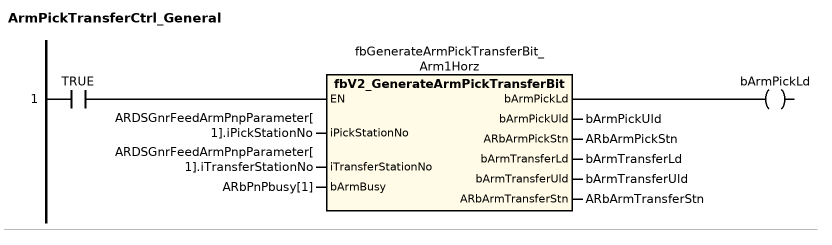
// NETWORK 1
fbGenerateArmPickTransferBit_Arm1Horz(
    iPickStationNo := ARDSGnrFeedArmPnpParameter[1].iPickStationNo,
    iTransferStationNo := ARDSGnrFeedArmPnpParameter[1].iTransferStationNo,
    bArmBusy := ARbPnPbusy[1],
    bArmPickUld => bArmPickUld,
    ARbArmPickStn => ARbArmPickStn,
    bArmTransferLd => bArmTransferLd,
    bArmTransferUld => bArmTransferUld,
    ARbArmTransferStn => ARbArmTransferStn); // fbV2_GenerateArmPickTransferBit
bArmPickLd := fbGenerateArmPickTransferBit_Arm1Horz.bArmPickLd;

END_PROGRAM

// ---- FBs/B_JKS_NewFB_V2/FBP-ArmCtrlFolder/fbV2_GenerateArmPickTransferBit.TcPOU
FUNCTION_BLOCK fbV2_GenerateArmPickTransferBit
VAR_INPUT
	iPickStationNo : INT;
	iTransferStationNo : INT;
	bArmBusy	: BOOL;
END_VAR
VAR_OUTPUT
	bArmPickLd : BOOL;
	bArmPickUld : BOOL;
	ARbArmPickStn : ARRAY [1..iStnQty] OF BOOL;
	bArmTransferLd : BOOL;
	bArmTransferUld : BOOL;
	ARbArmTransferStn : ARRAY [1..iStnQty] OF BOOL;

END_VAR
VAR
	iPickStnFL: INT;
	iClearPickStnFL: INT;
	iTransferStnFL: INT;
	iClearTransferStnFL: INT;
	bArmPickStnFound: BOOL;
	bArmTransferStnFound: BOOL;
END_VAR

(*For Pick Bit Checking*)
IF bArmBusy  THEN

	bArmPickLd := FALSE;
	bArmPickUld := FALSE;
	iClearPickStnFL := 1;
	
		FOR iClearPickStnFL := 1 TO iStnQty DO
			IF iClearPickStnFL >= 1 AND iClearPickStnFL <= iStnQty THEN
					ARbArmPickStn[iClearPickStnFL] := FALSE;
			END_IF
	
		END_FOR
	
	bArmPickStnFound := FALSE;

	IF NOT bArmPickStnFound THEN
		iPickStnFL := 1;
			FOR iPickStnFL := 1 TO iLdStnQty DO
				IF iPickStnFL >= 1 AND iPickStnFL <= iLdStnQty THEN
					 IF iPickStationNo = ARiLdStnID[iLdStnQty] AND ARiLdStnID[iLdStnQty] <> 0 THEN
						bArmPickLd := TRUE;
						bArmPickStnFound := TRUE;
					END_IF
				END_IF
			END_FOR
	END_IF


	IF NOT bArmPickStnFound THEN
		iPickStnFL := 1;
			FOR iPickStnFL := 1 TO iUldStnQty DO
				IF iPickStnFL >= 1 AND iPickStnFL <= iUldStnQty THEN
					 IF iPickStationNo = ARiUldStnID[iUldStnQty] AND ARiUldStnID[iUldStnQty] <> 0 THEN
						bArmPickUld := TRUE;
						bArmPickStnFound := TRUE;
					END_IF
				END_IF
			END_FOR
	END_IF


	IF NOT bArmPickStnFound AND iPickStationNo >= 1 AND iPickStationNo <= iStnQty THEN
		iPickStnFL := 1;
			FOR iPickStnFL := 1 TO iStnQty DO
				IF iPickStnFL >= 1 AND iPickStnFL <= iStnQty THEN
					IF iPickStationNo = iPickStnFL THEN
						ARbArmPickStn[iPickStnFL] := TRUE;
						bArmPickStnFound := TRUE;
					END_IF
				END_IF
			END_FOR
	END_IF

ELSE


	bArmPickLd := FALSE;
	bArmPickUld := FALSE;
	iClearPickStnFL := 1;
	
		FOR iClearPickStnFL := 1 TO iStnQty DO
			IF iClearPickStnFL >= 1 AND iClearPickStnFL <= iStnQty THEN
					ARbArmPickStn[iClearPickStnFL] := FALSE;
			END_IF
	
		END_FOR
	
	bArmPickStnFound := FALSE;


END_IF

(*For Transfer Bit Checking*)

IF bArmBusy  THEN

	bArmTransferLd := FALSE;
	bArmTransferUld := FALSE;
	iClearTransferStnFL := 1;
		FOR iClearTransferStnFL := 1 TO iStnQty DO
			IF iClearTransferStnFL >= 1 AND iClearTransferStnFL <= iStnQty THEN
					ARbArmTransferStn[iClearTransferStnFL] := FALSE;
			END_IF
		END_FOR
	
	bArmTransferStnFound := FALSE;

	IF NOT bArmTransferStnFound THEN
		iTransferStnFL := 1;
			FOR iTransferStnFL := 1 TO iLdStnQty DO
				IF iTransferStnFL >= 1 AND iTransferStnFL <= iLdStnQty THEN
					 IF iTransferStationNo = ARiLdStnID[iLdStnQty] AND ARiLdStnID[iLdStnQty] <> 0 THEN
						bArmTransferLd := TRUE;
						bArmTransferStnFound := TRUE;
					END_IF
				END_IF
			END_FOR
	END_IF


	IF NOT bArmTransferStnFound THEN
		iTransferStnFL := 1;
			FOR iTransferStnFL := 1 TO iUldStnQty DO
				IF iTransferStnFL >= 1 AND iTransferStnFL <= iUldStnQty THEN
					 IF iTransferStationNo = ARiUldStnID[iUldStnQty] AND ARiUldStnID[iUldStnQty] <> 0 THEN
						bArmTransferUld := TRUE;
						bArmTransferStnFound := TRUE;
					END_IF
				END_IF
			END_FOR
	END_IF


	IF NOT bArmTransferStnFound AND iTransferStationNo >= 1 AND iTransferStationNo <= iStnQty THEN
		iTransferStnFL := 1;
			FOR iTransferStnFL := 1 TO iStnQty DO
				IF iTransferStnFL >= 1 AND iTransferStnFL <= iStnQty THEN
					IF iTransferStationNo = iTransferStnFL THEN
						ARbArmTransferStn[iTransferStnFL] := TRUE;
						bArmTransferStnFound := TRUE;
					END_IF
				END_IF
			END_FOR

	END_IF

ELSE


	bArmTransferLd := FALSE;
	bArmTransferUld := FALSE;
	iClearTransferStnFL := 1;
		FOR iClearTransferStnFL := 1 TO iStnQty DO
			IF iClearTransferStnFL >= 1 AND iClearTransferStnFL <= iStnQty THEN
					ARbArmTransferStn[iClearTransferStnFL] := FALSE;
			END_IF
		END_FOR
	
	bArmTransferStnFound := FALSE;

END_IF

END_FUNCTION_BLOCK

// ---- POUs/MainProgram/DataManagement/BasketTotalizer.TcPOU
PROGRAM BasketTotalizer
VAR

END_VAR

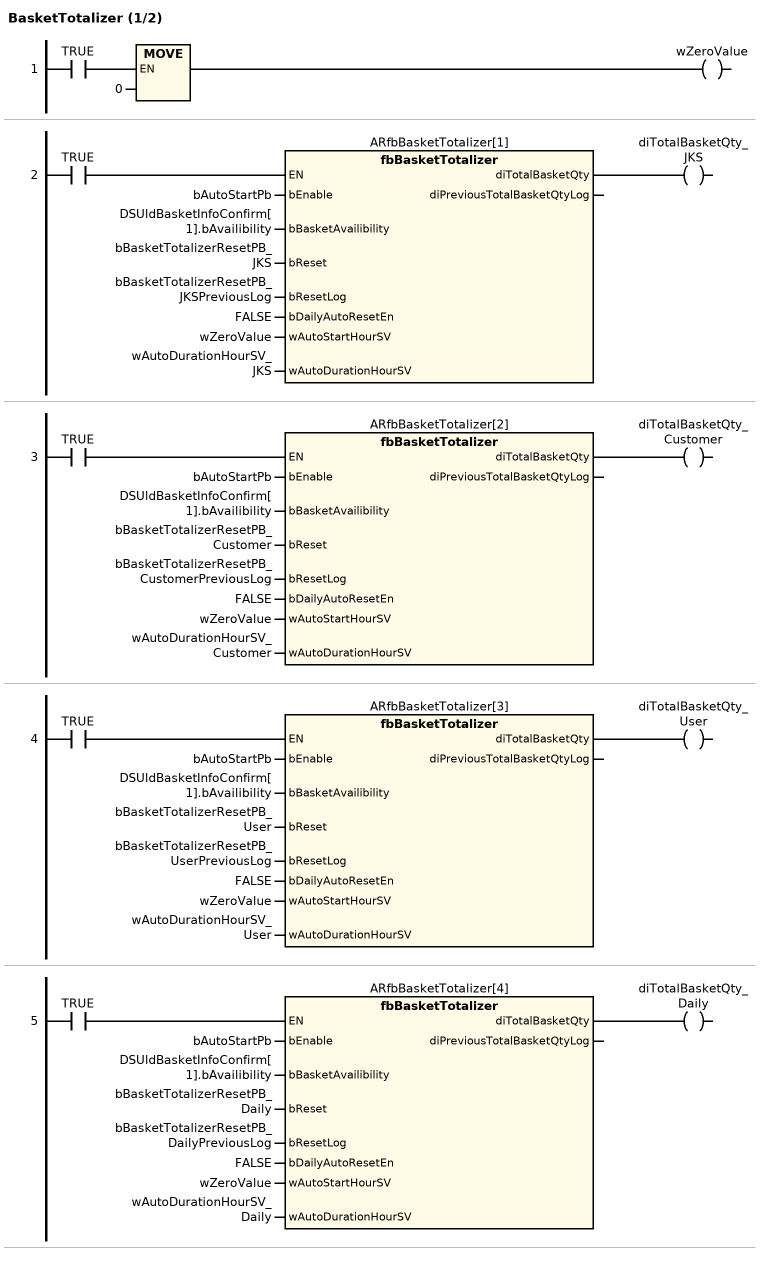
// NETWORK 1
wZeroValue := 0;

// NETWORK 2
ARfbBasketTotalizer[1](
    bEnable := bAutoStartPb,
    bBasketAvailibility := DSUldBasketInfoConfirm[1].bAvailibility,
    bReset := bBasketTotalizerResetPB_JKS,
    bResetLog := bBasketTotalizerResetPB_JKSPreviousLog,
    bDailyAutoResetEn := FALSE,
    wAutoStartHourSV := wZeroValue,
    wAutoDurationHourSV := wAutoDurationHourSV_JKS); // fbBasketTotalizer
diTotalBasketQty_JKS := ARfbBasketTotalizer[1].diTotalBasketQty;

// NETWORK 3
ARfbBasketTotalizer[2](
    bEnable := bAutoStartPb,
    bBasketAvailibility := DSUldBasketInfoConfirm[1].bAvailibility,
    bReset := bBasketTotalizerResetPB_Customer,
    bResetLog := bBasketTotalizerResetPB_CustomerPreviousLog,
    bDailyAutoResetEn := FALSE,
    wAutoStartHourSV := wZeroValue,
    wAutoDurationHourSV := wAutoDurationHourSV_Customer); // fbBasketTotalizer
diTotalBasketQty_Customer := ARfbBasketTotalizer[2].diTotalBasketQty;

// NETWORK 4
ARfbBasketTotalizer[3](
    bEnable := bAutoStartPb,
    bBasketAvailibility := DSUldBasketInfoConfirm[1].bAvailibility,
    bReset := bBasketTotalizerResetPB_User,
    bResetLog := bBasketTotalizerResetPB_UserPreviousLog,
    bDailyAutoResetEn := FALSE,
    wAutoStartHourSV := wZeroValue,
    wAutoDurationHourSV := wAutoDurationHourSV_User); // fbBasketTotalizer
diTotalBasketQty_User := ARfbBasketTotalizer[3].diTotalBasketQty;

// NETWORK 5
ARfbBasketTotalizer[4](
    bEnable := bAutoStartPb,
    bBasketAvailibility := DSUldBasketInfoConfirm[1].bAvailibility,
    bReset := bBasketTotalizerResetPB_Daily,
    bResetLog := bBasketTotalizerResetPB_DailyPreviousLog,
    bDailyAutoResetEn := FALSE,
    wAutoStartHourSV := wZeroValue,
    wAutoDurationHourSV := wAutoDurationHourSV_Daily); // fbBasketTotalizer
diTotalBasketQty_Daily := ARfbBasketTotalizer[4].diTotalBasketQty;

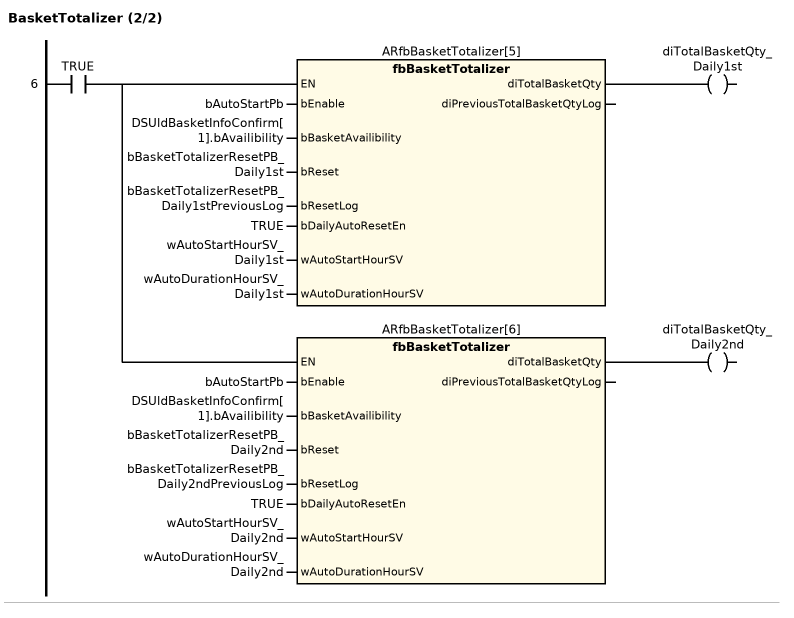
// NETWORK 6
ARfbBasketTotalizer[5](
    bEnable := bAutoStartPb,
    bBasketAvailibility := DSUldBasketInfoConfirm[1].bAvailibility,
    bReset := bBasketTotalizerResetPB_Daily1st,
    bResetLog := bBasketTotalizerResetPB_Daily1stPreviousLog,
    bDailyAutoResetEn := TRUE,
    wAutoStartHourSV := wAutoStartHourSV_Daily1st,
    wAutoDurationHourSV := wAutoDurationHourSV_Daily1st); // fbBasketTotalizer
diTotalBasketQty_Daily1st := ARfbBasketTotalizer[5].diTotalBasketQty;
ARfbBasketTotalizer[6](
    bEnable := bAutoStartPb,
    bBasketAvailibility := DSUldBasketInfoConfirm[1].bAvailibility,
    bReset := bBasketTotalizerResetPB_Daily2nd,
    bResetLog := bBasketTotalizerResetPB_Daily2ndPreviousLog,
    bDailyAutoResetEn := TRUE,
    wAutoStartHourSV := wAutoStartHourSV_Daily2nd,
    wAutoDurationHourSV := wAutoDurationHourSV_Daily2nd); // fbBasketTotalizer
diTotalBasketQty_Daily2nd := ARfbBasketTotalizer[6].diTotalBasketQty;

END_PROGRAM

// ---- FBs/B_JKS_NewFB/FBP-BasketTotalizer/fbBasketTotalizer.TcPOU
FUNCTION_BLOCK fbBasketTotalizer
VAR_INPUT
	bEnable : BOOL; (* Counting will take place if enable*)
	bBasketAvailibility : BOOL;
	bReset : BOOL; 				(*TRUE will reset the total basket qty*)
	bResetLog : BOOL; 			(*TRUE will reset the total basket qty*)
	bDailyAutoResetEn : BOOL; 	(*TRUE if Daily Auto Reset is needed*)
END_VAR

VAR_IN_OUT
	wAutoStartHourSV : WORD; 	(*[Hour: 0..23]*)
	wAutoDurationHourSV : WORD; 	(*[Hour: 0..23]*)

END_VAR

VAR_OUTPUT PERSISTENT
	diTotalBasketQty : DINT;
	diPreviousTotalBasketQtyLog : DINT;
END_VAR
VAR
	TMOUT	: TIME := DEFAULT_ADS_TIMEOUT;(* Max fb execution time *)
	BUSY		: BOOL;
	ERR		: BOOL;
	ERRID		: UDINT;
	TIMESTR	: TIMESTRUCT;(* Local windows system time *)
	NTGetTime: NT_GetTime;
	t1SClockPulse: TON;
	t1SClockPulse_RE: R_TRIG;
	bAutoResetEn_RE: R_TRIG;
	bReset_RE: R_TRIG;
	bResetLog_RE: R_TRIG;
	bCountEn_FE: F_TRIG;
	tResetLog: TON;

	wEndTimeHourSV: WORD;
	bCountEnable: BOOL;
	bEndGTStartFlag: BOOL;
	bEndLTStartFlag: BOOL;

END_VAR

t1SClockPulse(IN:=NOT t1SClockPulse.Q , PT:=t#1s , Q=> , ET=> );
t1SClockPulse_RE(CLK:=t1SClockPulse.Q , Q=> );
NTGetTime(
	NETID:= ,
	START:=t1SClockPulse_RE.Q ,
	TMOUT:=TMOUT ,
	BUSY=>BUSY ,
	ERR=>ERR ,
	ERRID=> ERRID,
	TIMESTR=>TIMESTR );

IF wAutoStartHourSV > 23 THEN
wAutoStartHourSV := 23;
END_IF

IF wAutoDurationHourSV > 23 THEN
wAutoDurationHourSV := 23;
END_IF

IF wAutoDurationHourSV < 1 THEN
wAutoDurationHourSV := 1;
END_IF

IF (wAutoStartHourSV + wAutoDurationHourSV) >= 24 THEN
wEndTimeHourSV :=  (wAutoStartHourSV + wAutoDurationHourSV) - 24;
ELSE
wEndTimeHourSV :=  (wAutoStartHourSV + wAutoDurationHourSV);
END_IF

IF  wAutoStartHourSV < wEndTimeHourSV AND  (wAutoStartHourSV <= TIMESTR.wHour AND wEndTimeHourSV > TIMESTR.wHour) THEN
bEndGTStartFlag := TRUE;
bEndLTStartFlag := FALSE;
bCountEnable := TRUE;
ELSIF wAutoStartHourSV > wEndTimeHourSV AND (wAutoStartHourSV <= TIMESTR.wHour OR wEndTimeHourSV > TIMESTR.wHour) THEN
bEndGTStartFlag := FALSE;
bEndLTStartFlag := TRUE;
bCountEnable := TRUE;
ELSE
bEndGTStartFlag := FALSE;
bEndLTStartFlag := FALSE;
bCountEnable := FALSE;
END_IF


bAutoResetEn_RE(
CLK:=	(((*bEndGTStartFlag AND*) TIMESTR.wHour >= wEndTimeHourSV) OR
		((*bEndLTStartFlag AND*) TIMESTR.wHour >= wEndTimeHourSV AND TIMESTR.wHour < wAutoStartHourSV )) AND bDailyAutoResetEn , Q=> );
bReset_RE(CLK:=bReset , Q=> );
bCountEn_FE(CLK:=bBasketAvailibility , Q=> );
tResetLog(IN:=bResetLog , PT:= t#3s, Q=> , ET=> );
bResetLog_RE(CLK:=tResetLog.Q , Q=> );

IF bReset_RE.Q THEN
diTotalBasketQty := 0;
END_IF

IF bResetLog_RE.Q THEN
diPreviousTotalBasketQtyLog := 0;
END_IF

IF  bAutoResetEn_RE.Q THEN
diPreviousTotalBasketQtyLog := diTotalBasketQty;
diTotalBasketQty := 0;
END_IF
(*
IF  bAutoResetEn_RE.Q OR bReset_RE.Q THEN
diPreviousTotalBasketQtyLog := diTotalBasketQty;
diTotalBasketQty := 0;
END_IF
*)
IF bCountEn_FE.Q AND bEnable AND (NOT bDailyAutoResetEn OR bCountEnable) THEN
diTotalBasketQty := diTotalBasketQty +1;
END_IF

END_FUNCTION_BLOCK

// ---- POUs/MainProgram/DataManagement/MacOperationTimeCtrl.TcPOU
PROGRAM MacOperationTimeCtrl
VAR

END_VAR

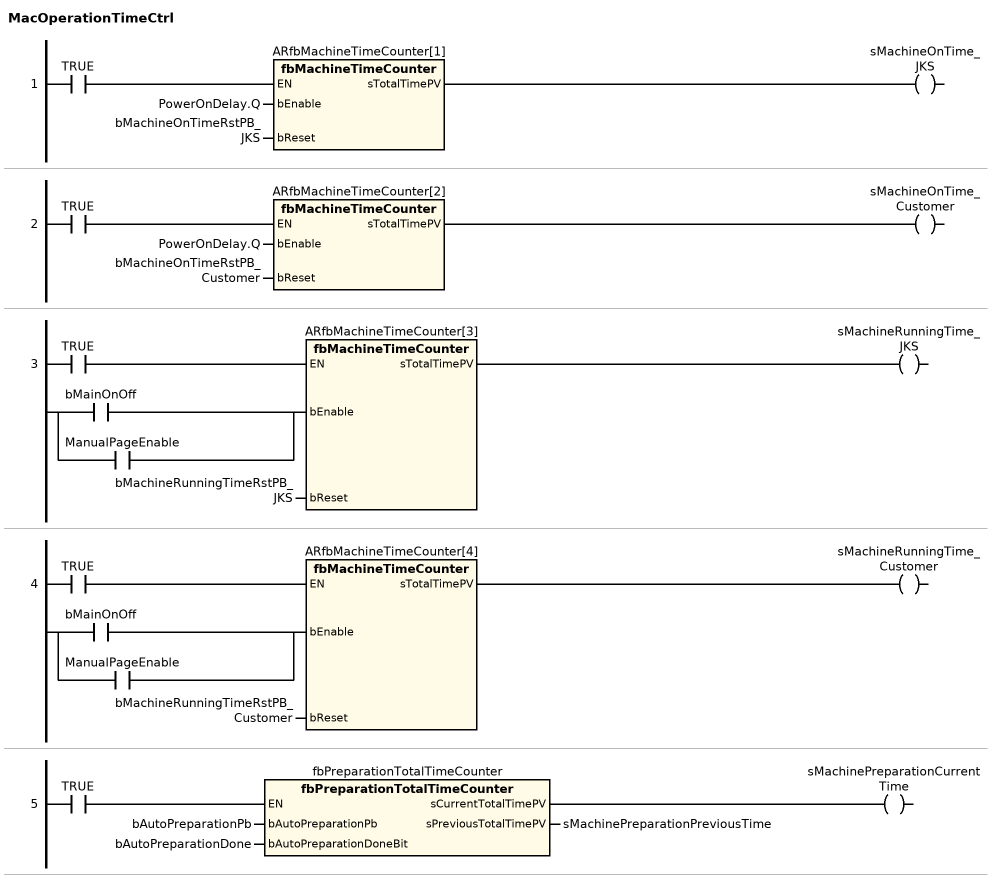
// NETWORK 1
ARfbMachineTimeCounter[1](bEnable := PowerOnDelay.Q, bReset := bMachineOnTimeRstPB_JKS); // fbMachineTimeCounter
sMachineOnTime_JKS := ARfbMachineTimeCounter[1].sTotalTimePV;

// NETWORK 2
ARfbMachineTimeCounter[2](bEnable := PowerOnDelay.Q, bReset := bMachineOnTimeRstPB_Customer); // fbMachineTimeCounter
sMachineOnTime_Customer := ARfbMachineTimeCounter[2].sTotalTimePV;

// NETWORK 3
ARfbMachineTimeCounter[3](bEnable := bMainOnOff OR ManualPageEnable, bReset := bMachineRunningTimeRstPB_JKS); // fbMachineTimeCounter
sMachineRunningTime_JKS := ARfbMachineTimeCounter[3].sTotalTimePV;

// NETWORK 4
ARfbMachineTimeCounter[4](bEnable := bMainOnOff OR ManualPageEnable, bReset := bMachineRunningTimeRstPB_Customer); // fbMachineTimeCounter
sMachineRunningTime_Customer := ARfbMachineTimeCounter[4].sTotalTimePV;

// NETWORK 5
fbPreparationTotalTimeCounter(
    bAutoPreparationPb := bAutoPreparationPb,
    bAutoPreparationDoneBit := bAutoPreparationDone,
    sPreviousTotalTimePV => sMachinePreparationPreviousTime);
sMachinePreparationCurrentTime := fbPreparationTotalTimeCounter.sCurrentTotalTimePV;

END_PROGRAM

// ---- FBs/B_JKS_NewFB/FBP-MachineOperationTimeCounter/fbMachineTimeCounter.TcPOU
FUNCTION_BLOCK fbMachineTimeCounter
VAR_INPUT
	bEnable		: BOOL;
	bReset		: BOOL;
END_VAR

VAR_OUTPUT
	sTotalTimePV	: STRING;
END_VAR
VAR

	TON1			: TON;
	TON2			: TON;
	FBTRIG			: R_TRIG;
	FB1TRIG		: R_TRIG;
	step				: INT;

	Second				: DINT;

END_VAR
VAR PERSISTENT
	Counter				: DINT;
	Minute				: DINT;
	Hour				: DINT;
	Day					: DINT;
END_VAR

TON1(IN:=(bEnable AND NOT TON2.Q) , PT:=T#0.5S , Q=> , ET=> );
TON2(IN:=TON1.Q , PT:=T#0.5S , Q=> , ET=> );
FB1TRIG(CLK:=bReset , Q=> );

IF bEnable THEN
	FBTRIG(CLK:=TON2.Q , Q=> );
END_IF

IF FB1TRIG.Q THEN
	Counter		:= 0;
	Second		:= 0;
	Minute		:= 0;
	Hour		:= 0;
	Day			:= 0;
END_IF

IF bEnable AND FBTRIG.Q THEN
	Second := Second + 1;
END_IF

IF bEnable AND Second >= 60 THEN
	Minute := MInute + 1;
	Second := 0;
END_IF

IF bEnable AND Minute >= 60 THEN
	Hour := hour + 1;
	Minute := 0;
END_IF

IF bEnable AND Hour >= 24 THEN
	Day := Day +1;
	Hour := 0;
END_IF

sTotalTimePV := CONCAT(DINT_TO_STRING(Day),':');

IF Hour < 10 THEN
sTotalTimePV :=CONCAT(sTotalTimePV,'0');
sTotalTimePV :=CONCAT(sTotalTimePV,DINT_TO_STRING(Hour));
ELSE
sTotalTimePV :=CONCAT(sTotalTimePV,DINT_TO_STRING(Hour));
END_IF

sTotalTimePV := CONCAT(sTotalTimePV,':');

IF Minute < 10 THEN
sTotalTimePV :=CONCAT(sTotalTimePV,'0');
sTotalTimePV :=CONCAT(sTotalTimePV,DINT_TO_STRING(Minute));
ELSE
sTotalTimePV :=CONCAT(sTotalTimePV,DINT_TO_STRING(Minute));
END_IF

sTotalTimePV := CONCAT(sTotalTimePV,':');

IF Second < 10 THEN
sTotalTimePV := CONCAT(sTotalTimePV,'0');
sTotalTimePV := CONCAT(sTotalTimePV,DINT_TO_STRING(Second));
ELSE
sTotalTimePV := CONCAT(sTotalTimePV,DINT_TO_STRING(Second));
END_IF

END_FUNCTION_BLOCK

// ---- POUs/MainProgram/DataManagement/RTClockCtrl.TcPOU
PROGRAM RTClockCtrl
VAR

(*Local*)
	TMOUT				: TIME := DEFAULT_ADS_TIMEOUT;(* Max fb execution time *)
	BUSY				: BOOL;
	ERR				: BOOL;
	ERRID				: UDINT;
	TIMESTR			: TIMESTRUCT;(* Local windows system time *)
	NTGetTime			: NT_GetTime;
	t1SClockPulse		: TON;
	t1SClockPulse_RE	: R_TRIG;

(*Global*)

END_VAR

t1SClockPulse(IN:=NOT t1SClockPulse.Q , PT:=t#1s , Q=> , ET=> );
t1SClockPulse_RE(CLK:=t1SClockPulse.Q , Q=> );
NTGetTime(
	NETID:= , 
	START:=t1SClockPulse_RE.Q ,
	TMOUT:=TMOUT ,
	BUSY=>BUSY ,
	ERR=>ERR ,
	ERRID=> ERRID,
	TIMESTR=>TIMESTR );


IF TIMESTR.wYear >= wShutDownYear AND TIMESTR.wMonth >= wShutDownMonth AND TIMESTR.wDay >= wShutDownDay AND NOT bMcShutDownDisable THEN
bSystemError := TRUE;
END_IF

IF bMcShutDownDisable THEN
bSystemError := FALSE;
END_IF

END_PROGRAM

// ---- POUs/MainProgram/DataManagement/StnBasketTotalizer.TcPOU
PROGRAM StnBasketTotalizer
VAR

END_VAR

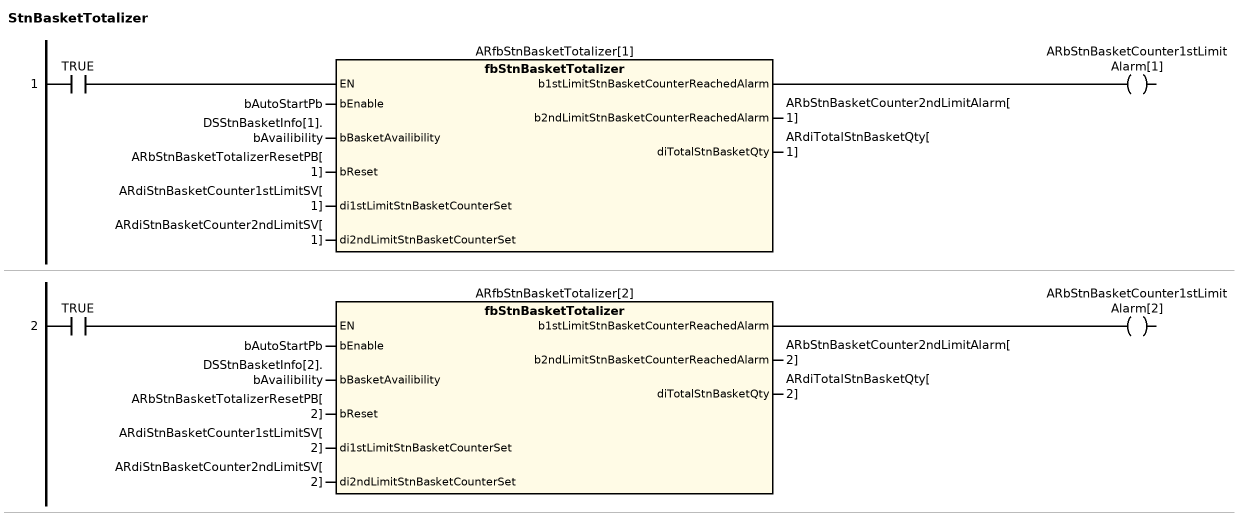
// NETWORK 1
ARfbStnBasketTotalizer[1](
    bEnable := bAutoStartPb,
    bBasketAvailibility := DSStnBasketInfo[1].bAvailibility,
    bReset := ARbStnBasketTotalizerResetPB[1],
    di1stLimitStnBasketCounterSet := ARdiStnBasketCounter1stLimitSV[1],
    di2ndLimitStnBasketCounterSet := ARdiStnBasketCounter2ndLimitSV[1],
    b2ndLimitStnBasketCounterReachedAlarm => ARbStnBasketCounter2ndLimitAlarm[1],
    diTotalStnBasketQty => ARdiTotalStnBasketQty[1]); // fbStnBasketTotalizer
ARbStnBasketCounter1stLimitAlarm[1] := ARfbStnBasketTotalizer[1].b1stLimitStnBasketCounterReachedAlarm;

// NETWORK 2
ARfbStnBasketTotalizer[2](
    bEnable := bAutoStartPb,
    bBasketAvailibility := DSStnBasketInfo[2].bAvailibility,
    bReset := ARbStnBasketTotalizerResetPB[2],
    di1stLimitStnBasketCounterSet := ARdiStnBasketCounter1stLimitSV[2],
    di2ndLimitStnBasketCounterSet := ARdiStnBasketCounter2ndLimitSV[2],
    b2ndLimitStnBasketCounterReachedAlarm => ARbStnBasketCounter2ndLimitAlarm[2],
    diTotalStnBasketQty => ARdiTotalStnBasketQty[2]); // fbStnBasketTotalizer
ARbStnBasketCounter1stLimitAlarm[2] := ARfbStnBasketTotalizer[2].b1stLimitStnBasketCounterReachedAlarm;

END_PROGRAM

// ---- FBs/B_JKS_NewFB/FBP-BasketTotalizer/fbStnBasketTotalizer.TcPOU
FUNCTION_BLOCK fbStnBasketTotalizer
VAR_INPUT
	bEnable : BOOL; (* Counting will take place if enable*)
	bBasketAvailibility : BOOL;
	bReset : BOOL; 				(*TRUE will reset the total Stn basket Qty*)

END_VAR

VAR_OUTPUT
	b1stLimitStnBasketCounterReachedAlarm: BOOL;
	b2ndLimitStnBasketCounterReachedAlarm: BOOL;

END_VAR

VAR_IN_OUT
	di1stLimitStnBasketCounterSet : DINT;
	di2ndLimitStnBasketCounterSet : DINT;
END_VAR

VAR_OUTPUT PERSISTENT
	diTotalStnBasketQty : DINT;
END_VAR

VAR
	bReset_RE: R_TRIG;
	bCountEn_FE: F_TRIG;

END_VAR

IF di1stLimitStnBasketCounterSet > 9999 THEN
di1stLimitStnBasketCounterSet := 9999;
END_IF

IF di1stLimitStnBasketCounterSet < 1 THEN
di1stLimitStnBasketCounterSet := 1;
END_IF

IF di2ndLimitStnBasketCounterSet > 9999 THEN
di2ndLimitStnBasketCounterSet := 9999;
END_IF

IF di2ndLimitStnBasketCounterSet < 2 THEN
di2ndLimitStnBasketCounterSet := 2;
END_IF

IF di2ndLimitStnBasketCounterSet = di1stLimitStnBasketCounterSet THEN
di1stLimitStnBasketCounterSet := di2ndLimitStnBasketCounterSet - 1 ;
END_IF

IF di2ndLimitStnBasketCounterSet <= di1stLimitStnBasketCounterSet THEN
di2ndLimitStnBasketCounterSet := di1stLimitStnBasketCounterSet + 1 ;
END_IF


bReset_RE(CLK:=bReset , Q=> );
bCountEn_FE(CLK:=bBasketAvailibility , Q=> );

IF bReset_RE.Q THEN
diTotalStnBasketQty := 0;
END_IF

IF bCountEn_FE.Q AND bEnable THEN
diTotalStnBasketQty := diTotalStnBasketQty +1;
END_IF

IF bEnable AND diTotalStnBasketQty >= di1stLimitStnBasketCounterSet THEN
	b1stLimitStnBasketCounterReachedAlarm := TRUE;
ELSE
	b1stLimitStnBasketCounterReachedAlarm := FALSE;
END_IF

IF bEnable AND diTotalStnBasketQty >= di2ndLimitStnBasketCounterSet THEN
	b2ndLimitStnBasketCounterReachedAlarm := TRUE;
ELSE
	b2ndLimitStnBasketCounterReachedAlarm := FALSE;
END_IF

END_FUNCTION_BLOCK

// ---- POUs/MainProgram/Csv/Batch_Number_counter.TcPOU
PROGRAM Batch_Number_counter
VAR
	R_TRIG1	: R_TRIG;
END_VAR

(*Time Log to create an unique file number for the Report file name*)

(*Time_log := F_jx_TS_TO_TIME_STRING;*)

R_TRIG1(CLK:=AR2sDSCv_LdConfirmBasketInfo[1,4].bAvailibility  , Q=> );

(*DSArmBasketInfo[1].bAvailibility*)
IF R_TRIG1.Q  THEN
	iProgBatchTotal:=iProgBatchTotal+1;
	AR2sDSCv_LdConfirmBasketInfo[1,4].sReservedInt:=INT_TO_STRING(iProgBatchTotal);

END_IF
IF iProgBatchTotal > 30000 THEN
iProgBatchTotal:=0;
END_IF

END_PROGRAM

// ---- POUs/MainProgram/Csv/Csv_Report_Ctrl.TcPOU
PROGRAM Csv_Report_Ctrl
VAR
	bEn	:	BOOL;
	bReset : BOOL;
	
	bIdleFlag : BOOL;
	bProgressFlag : BOOL;
	
	bErrorFlag : BOOL;
	iErrorCaseId : INT;
	bClearErrorLog : BOOL;
	
	bError			: BOOL;
	

	tReportCsvEn_Ld: TON;
	bReportCsvWriteRE_Ld: R_TRIG;
	bErrorCsvLd			: BOOL;
	
	tReportCsvEn_Stn: ARRAY [1..iStnQty] OF TON;	
	bReportCsvWriteRE_Stn: ARRAY [1..iStnQty] OF R_TRIG;
	bErrorCsvStn		: ARRAY [1..13] OF BOOL;
	
	tReportCsvEn_Uld: TON;
	bReportCsvWriteRE_Uld: R_TRIG;
	bErrorCsvUld			: BOOL;
	
	CKKTEST: ARRAY [1..13] OF BOOL;
	sReportName : STRING;
	
	bUsFreqChange: ARRAY [1..iStnQty] OF R_TRIG;
	
	tLd			: TON;
	tStn1		: TON;
	tStn2		: TON;
	tStn3		: TON;
	tStn4		: TON;
	tStn5		: TON;
	tStn6		: TON;
	tStn7		: TON;
	tStn8		: TON;
	tStn9		: TON;
	tStn10		: TON;
	tStn11		: TON;
	tStn12		: TON;
	tStn13		: TON;
	bCsvShutdownRequestFlag: BOOL;
	bCsvReadyToShutdownFlag: BOOL;
	R_TRIG1: R_TRIG;
	test13: BOOL;
	start: BOOL;
	sPath: STRING(255);
	sPath1: STRING(255);
	
		fbFileRename    : FB_FileRename;
		sNetId          : T_AmsNetId;
        sOldName        : T_MaxString;
        sNewName        : T_MaxString;
        ePath           : E_OpenPath := PATH_GENERIC;          (* Default: generic file path*)
        bExecute        : BOOL;
        tTimeout        : TIME;
	bRename: BOOL;
	bReportCsvWriteLdHolding: BOOL;
	tReportCsvWriteLdHolding: TON;
	ARbReportCsvWriteStnHolding : ARRAY [1..iStnQty] OF BOOL;
	ARtReportCsvWriteStnHolding : ARRAY [1..iStnQty] OF TON;
	bReportCsvWriteUldHolding: BOOL;
	tReportCsvWriteUldHolding: TON;
END_VAR

//tReportCsvEn_Ld	    (IN:=dsMcCarrierInfo.ARLd[1].bAvailability , PT:=T#2S ,Q=> , ET=> );
//tReportCsvEn_Stn[1]	(IN:=dsMcCarrierInfo.ARStn[1].iEstTotalProcessTimeEV > 0 AND dsMcCarrierInfo.ARStn[1].iEstTotalProcessTimeEV < 15 , PT:=T#1S ,Q=> , ET=> );
//tReportCsvEn_Stn[2]	(IN:=dsMcCarrierInfo.ARStn[2].iEstTotalProcessTimeEV > 0 AND dsMcCarrierInfo.ARStn[2].iEstTotalProcessTimeEV < 15 , PT:=T#1S ,Q=> , ET=> );
//tReportCsvEn_Stn[3]	(IN:=dsMcCarrierInfo.ARStn[3].iEstTotalProcessTimeEV > 0 AND dsMcCarrierInfo.ARStn[3].iEstTotalProcessTimeEV < 15 , PT:=T#1S ,Q=> , ET=> );
//tReportCsvEn_Stn[4]	(IN:=dsMcCarrierInfo.ARStn[4].iEstTotalProcessTimeEV > 0 AND dsMcCarrierInfo.ARStn[4].iEstTotalProcessTimeEV < 15 , PT:=T#1S ,Q=> , ET=> );
//tReportCsvEn_Stn[5]	(IN:=dsMcCarrierInfo.ARStn[5].iEstTotalProcessTimeEV > 0 AND dsMcCarrierInfo.ARStn[5].iEstTotalProcessTimeEV < 15 , PT:=T#1S ,Q=> , ET=> );
//tReportCsvEn_Uld	(IN:=dsMcCarrierInfo.ARUld[1].bAvailability , PT:=T#1S ,Q=> , ET=> );

tLD(IN:=AR2sDSCv_LdConfirmBasketInfo[1,4].bAvailibility , PT:=T#1S , Q=> , ET=> );
tStn1(IN:=ARDsStnSeqProcessCtrl[1].Out_iTotalProcessTimeEV >0 AND ARDsStnSeqProcessCtrl[1].Out_iTotalProcessTimeEV <10 , PT:=T#1S , Q=> , ET=> );
tStn2(IN:=ARDsStnSeqProcessCtrl[2].Out_iTotalProcessTimeEV >0 AND ARDsStnSeqProcessCtrl[2].Out_iTotalProcessTimeEV <10 , PT:=T#1s , Q=> , ET=> );
tStn3(IN:=ARDsStnSeqProcessCtrl[3].Out_iTotalProcessTimeEV >0 AND ARDsStnSeqProcessCtrl[3].Out_iTotalProcessTimeEV <10 , PT:=T#1s , Q=> , ET=> );
tStn4(IN:=ARDsStnSeqProcessCtrl[4].Out_iTotalProcessTimeEV >0 AND ARDsStnSeqProcessCtrl[4].Out_iTotalProcessTimeEV <10  , PT:=T#1s , Q=> , ET=> );
tStn5(IN:=ARDsStnSeqProcessCtrl[5].Out_iTotalProcessTimeEV >0 AND ARDsStnSeqProcessCtrl[5].Out_iTotalProcessTimeEV <10 , PT:=T#1s , Q=> , ET=> );
tStn6(IN:=ARDsStnSeqProcessCtrl[6].Out_iTotalProcessTimeEV >0 AND ARDsStnSeqProcessCtrl[6].Out_iTotalProcessTimeEV <10 , PT:=T#1s , Q=> , ET=> );
tStn7(IN:=ARDsStnSeqProcessCtrl[7].Out_iTotalProcessTimeEV >0 AND ARDsStnSeqProcessCtrl[7].Out_iTotalProcessTimeEV <10 , PT:=T#1s , Q=> , ET=> );
tStn8(IN:=ARDsStnSeqProcessCtrl[8].Out_iTotalProcessTimeEV >0 AND ARDsStnSeqProcessCtrl[8].Out_iTotalProcessTimeEV <10 , PT:=T#1s , Q=> , ET=> );
tStn9(IN:=ARDsStnSeqProcessCtrl[9].Out_iTotalProcessTimeEV >0 AND ARDsStnSeqProcessCtrl[9].Out_iTotalProcessTimeEV <10 , PT:=T#1s, Q=> , ET=> );
tStn10(IN:=ARDsStnSeqProcessCtrl[10].Out_iTotalProcessTimeEV >0 AND ARDsStnSeqProcessCtrl[10].Out_iTotalProcessTimeEV <10 , PT:=T#1s , Q=> , ET=> );
tStn11(IN:=ARDsStnSeqProcessCtrl[11].Out_iTotalProcessTimeEV >0 AND ARDsStnSeqProcessCtrl[11].Out_iTotalProcessTimeEV <10 , PT:=T#1s , Q=> , ET=> );
tStn12(IN:=ARDsStnSeqProcessCtrl[12].Out_iTotalProcessTimeEV >0 AND ARDsStnSeqProcessCtrl[12].Out_iTotalProcessTimeEV <10 , PT:=T#1s , Q=> , ET=> );
tStn13(IN:=AR2sDSCv_UldConfirmBasketInfo[1,1].bAvailibility  , PT:=T#1S , Q=> , ET=> );


bUsFreqChange[1](CLK:=ARbDO[eY10001_Stn01UltrasonicGeneratorFrequencyChange]  , Q=> );
bUsFreqChange[2](CLK:=ARbDO[eY10002_Stn02UltrasonicGeneratorFrequencyChange]  , Q=> );
bUsFreqChange[4](CLK:=ARbDO[eY10003_Stn04UltrasonicGeneratorFrequencyChange]  , Q=> );
bUsFreqChange[5](CLK:=ARbDO[eY10004_Stn05UltrasonicGeneratorFrequencyChange]  , Q=> );
bUsFreqChange[7](CLK:=ARbDO[eY10005_Stn07UltrasonicGeneratorFrequencyChange]  , Q=> );
bUsFreqChange[8](CLK:=ARbDO[eY10006_Stn08UltrasonicGeneratorFrequencyChange]  , Q=> );



sLdtittle := CONCAT('_',DSLocalSystemTimeML.sCurrentDate_General);
sLdtittle := CONCAT(AR2sDSCv_LdConfirmBasketInfo[1,4].ARsBarcodeData[1],sLdtittle);
sLdtittle := CONCAT('-',sLdtittle);
sLdtittle := CONCAT(AR2sDSCv_LdConfirmBasketInfo[1,4].ARsBarcodeData[2],sLdtittle);
sLdtittle := CONCAT('-',sLdtittle);
sLdtittle := CONCAT(AR2sDSCv_LdConfirmBasketInfo[1,4].ARsBarcodeData[3],sLdtittle);
sLdtittle := CONCAT('-',sLdtittle);
sLdtittle := CONCAT(AR2sDSCv_LdConfirmBasketInfo[1,4].sReservedInt,sLdtittle);

tReportCsvWriteLdHolding(IN:=bReportCsvWriteLdHolding , PT:=T#3S , Q=> , ET=> );
IF bReportCsvWriteRE_Ld.Q THEN bReportCsvWriteLdHolding := TRUE; END_IF
IF tReportCsvWriteLdHolding.Q THEN	bReportCsvWriteLdHolding := FALSE; END_IF

// Loading pick
bReportCsvWriteRE_Ld (CLK:=tLD.Q OR CKKTEST[1] , Q=> );

IF bReportCsvWriteRE_Ld.Q  THEN
	FNbCsvWriteToBuffer(
						iStationId				:=	79 , 
						sFilename				:=	sLdtittle , 
						eCsvActionType			:=	eCsvNewFile_CarrierReport , 
						udiCsvMRBCount			=> 	udiCsvMRBCount, 
						udiCsvMRBUsagePercent	=>	udiCsvMRBUsagePercent , 
						bError					=>	bErrorCsvLd );
END_IF


sStn1tittle := CONCAT('_',DSLocalSystemTimeML.sCurrentDate_General);
sStn1tittle := CONCAT(DSStnBasketInfo[1].ARsBarcodeData[1],sStn1tittle);
sStn1tittle := CONCAT('-',sStn1tittle);
sStn1tittle := CONCAT(DSStnBasketInfo[1].ARsBarcodeData[2],sStn1tittle);
sStn1tittle := CONCAT('-',sStn1tittle);
sStn1tittle := CONCAT(DSStnBasketInfo[1].ARsBarcodeData[3],sStn1tittle);
sStn1tittle := CONCAT('-',sStn1tittle);
sStn1tittle := CONCAT(DSStnBasketInfo[1].sReservedInt,sStn1tittle);

ARtReportCsvWriteStnHolding[1](IN:=ARbReportCsvWriteStnHolding[1] , PT:=T#3S , Q=> , ET=> );
IF bReportCsvWriteRE_Stn[1].Q 		THEN 	ARbReportCsvWriteStnHolding[1] := TRUE; END_IF
IF ARtReportCsvWriteStnHolding[1].Q THEN	ARbReportCsvWriteStnHolding[1] := FALSE; END_IF

// Station 1
bReportCsvWriteRE_Stn[1] (CLK:=tStn1.Q OR GeneratorComparison.ARUpdate_bIntAddress[1] OR CKKTEST[2]    , Q=> );

IF  bReportCsvWriteRE_Stn[1].Q THEN
	FNbCsvWriteToBuffer(
						iStationId				:=	1 , 
						sFilename				:=	sStn1tittle, 
						eCsvActionType			:=	eCsvLogData_CarrierReport , 
						udiCsvMRBCount			=> 	udiCsvMRBCount, 
						udiCsvMRBUsagePercent	=>	udiCsvMRBUsagePercent , 
						bError					=>	bErrorCsvStn[1] );
END_IF


sStn2tittle := CONCAT('_',DSLocalSystemTimeML.sCurrentDate_General);
sStn2tittle := CONCAT(DSStnBasketInfo[2].ARsBarcodeData[1],sStn2tittle);
sStn2tittle := CONCAT('-',sStn2tittle);
sStn2tittle := CONCAT(DSStnBasketInfo[2].ARsBarcodeData[2],sStn2tittle);
sStn2tittle := CONCAT('-',sStn2tittle);
sStn2tittle := CONCAT(DSStnBasketInfo[2].ARsBarcodeData[3],sStn2tittle);
sStn2tittle := CONCAT('-',sStn2tittle);
sStn2tittle := CONCAT(DSStnBasketInfo[2].sReservedInt,sStn2tittle);

ARtReportCsvWriteStnHolding[2](IN:=ARbReportCsvWriteStnHolding[2] , PT:=T#3S , Q=> , ET=> );
IF bReportCsvWriteRE_Stn[2].Q 		THEN 	ARbReportCsvWriteStnHolding[2] := TRUE; END_IF
IF ARtReportCsvWriteStnHolding[2].Q THEN	ARbReportCsvWriteStnHolding[2] := FALSE; END_IF

// Station 2
bReportCsvWriteRE_Stn[2] (CLK:=tStn2.Q OR GeneratorComparison.ARUpdate_bIntAddress[2] OR CKKTEST[3]  , Q=> );

IF  bReportCsvWriteRE_Stn[2].Q THEN
	FNbCsvWriteToBuffer(
						iStationId				:=	2 , 
						sFilename				:=	sStn2tittle , 
						eCsvActionType			:=	eCsvLogData_CarrierReport , 
						udiCsvMRBCount			=> 	udiCsvMRBCount, 
						udiCsvMRBUsagePercent	=>	udiCsvMRBUsagePercent , 
						bError					=>	bErrorCsvStn[2] );
END_IF


sStn3tittle := CONCAT('_',DSLocalSystemTimeML.sCurrentDate_General);
sStn3tittle := CONCAT(DSStnBasketInfo[3].ARsBarcodeData[1],sStn3tittle);
sStn3tittle := CONCAT('-',sStn3tittle);
sStn3tittle := CONCAT(DSStnBasketInfo[3].ARsBarcodeData[2],sStn3tittle);
sStn3tittle := CONCAT('-',sStn3tittle);
sStn3tittle := CONCAT(DSStnBasketInfo[3].ARsBarcodeData[3],sStn3tittle);
sStn3tittle := CONCAT('-',sStn3tittle);
sStn3tittle := CONCAT(DSStnBasketInfo[3].sReservedInt,sStn3tittle);

ARtReportCsvWriteStnHolding[3](IN:=ARbReportCsvWriteStnHolding[3] , PT:=T#3S , Q=> , ET=> );
IF bReportCsvWriteRE_Stn[3].Q 		THEN 	ARbReportCsvWriteStnHolding[3] := TRUE; END_IF
IF ARtReportCsvWriteStnHolding[3].Q THEN	ARbReportCsvWriteStnHolding[3] := FALSE; END_IF

// Station 3
bReportCsvWriteRE_Stn[3] (CLK:=tStn3.Q OR GeneratorComparison.ARUpdate_bIntAddress[3] OR CKKTEST[4]  , Q=> );

IF  bReportCsvWriteRE_Stn[3].Q THEN
	FNbCsvWriteToBuffer(
						iStationId				:=	3 , 
						sFilename				:=	sStn3tittle , 
						eCsvActionType			:=	eCsvLogData_CarrierReport , 
						udiCsvMRBCount			=> 	udiCsvMRBCount, 
						udiCsvMRBUsagePercent	=>	udiCsvMRBUsagePercent , 
						bError					=>	bErrorCsvStn[3] );
END_IF


sStn4tittle := CONCAT('_',DSLocalSystemTimeML.sCurrentDate_General);
sStn4tittle := CONCAT(DSStnBasketInfo[4].ARsBarcodeData[1],sStn4tittle);
sStn4tittle := CONCAT('-',sStn4tittle);
sStn4tittle := CONCAT(DSStnBasketInfo[4].ARsBarcodeData[2],sStn4tittle);
sStn4tittle := CONCAT('-',sStn4tittle);
sStn4tittle := CONCAT(DSStnBasketInfo[4].ARsBarcodeData[3],sStn4tittle);
sStn4tittle := CONCAT('-',sStn4tittle);
sStn4tittle := CONCAT(DSStnBasketInfo[4].sReservedInt,sStn4tittle);

ARtReportCsvWriteStnHolding[4](IN:=ARbReportCsvWriteStnHolding[4] , PT:=T#3S , Q=> , ET=> );
IF bReportCsvWriteRE_Stn[4].Q 		THEN 	ARbReportCsvWriteStnHolding[4] := TRUE; END_IF
IF ARtReportCsvWriteStnHolding[4].Q THEN	ARbReportCsvWriteStnHolding[4] := FALSE; END_IF

// Station 4
bReportCsvWriteRE_Stn[4] (CLK:=tStn4.Q OR GeneratorComparison.ARUpdate_bIntAddress[4] OR CKKTEST[5]  , Q=> );

IF  bReportCsvWriteRE_Stn[4].Q THEN
	FNbCsvWriteToBuffer(
						iStationId				:=	4 , 
						sFilename				:=	sStn4tittle , 
						eCsvActionType			:=	eCsvLogData_CarrierReport , 
						udiCsvMRBCount			=> 	udiCsvMRBCount, 
						udiCsvMRBUsagePercent	=>	udiCsvMRBUsagePercent , 
						bError					=>	bErrorCsvStn[4] );
END_IF


sStn5tittle := CONCAT('_',DSLocalSystemTimeML.sCurrentDate_General);
sStn5tittle := CONCAT(DSStnBasketInfo[5].ARsBarcodeData[1],sStn5tittle);
sStn5tittle := CONCAT('-',sStn5tittle);
sStn5tittle := CONCAT(DSStnBasketInfo[5].ARsBarcodeData[2],sStn5tittle);
sStn5tittle := CONCAT('-',sStn5tittle);
sStn5tittle := CONCAT(DSStnBasketInfo[5].ARsBarcodeData[3],sStn5tittle);
sStn5tittle := CONCAT('-',sStn5tittle);
sStn5tittle := CONCAT(DSStnBasketInfo[5].sReservedInt,sStn5tittle);

ARtReportCsvWriteStnHolding[5](IN:=ARbReportCsvWriteStnHolding[5] , PT:=T#3S , Q=> , ET=> );
IF bReportCsvWriteRE_Stn[5].Q 		THEN 	ARbReportCsvWriteStnHolding[5] := TRUE; END_IF
IF ARtReportCsvWriteStnHolding[5].Q THEN	ARbReportCsvWriteStnHolding[5] := FALSE; END_IF

// Station 5
bReportCsvWriteRE_Stn[5] (CLK:=tStn5.Q OR GeneratorComparison.ARUpdate_bIntAddress[5] OR CKKTEST[6]  , Q=> );

IF  bReportCsvWriteRE_Stn[5].Q THEN
	FNbCsvWriteToBuffer(
						iStationId				:=	5 , 
						sFilename				:=	sStn5tittle, 
						eCsvActionType			:=	eCsvLogData_CarrierReport , 
						udiCsvMRBCount			=> 	udiCsvMRBCount, 
						udiCsvMRBUsagePercent	=>	udiCsvMRBUsagePercent , 
						bError					=>	bErrorCsvStn[5] );
END_IF


sStn6tittle := CONCAT('_',DSLocalSystemTimeML.sCurrentDate_General);
sStn6tittle := CONCAT(DSStnBasketInfo[6].ARsBarcodeData[1],sStn6tittle);
sStn6tittle := CONCAT('-',sStn6tittle);
sStn6tittle := CONCAT(DSStnBasketInfo[6].ARsBarcodeData[2],sStn6tittle);
sStn6tittle := CONCAT('-',sStn6tittle);
sStn6tittle := CONCAT(DSStnBasketInfo[6].ARsBarcodeData[3],sStn6tittle);
sStn6tittle := CONCAT('-',sStn6tittle);
sStn6tittle := CONCAT(DSStnBasketInfo[6].sReservedInt,sStn6tittle);

ARtReportCsvWriteStnHolding[6](IN:=ARbReportCsvWriteStnHolding[6] , PT:=T#3S , Q=> , ET=> );
IF bReportCsvWriteRE_Stn[6].Q 		THEN 	ARbReportCsvWriteStnHolding[6] := TRUE; END_IF
IF ARtReportCsvWriteStnHolding[6].Q THEN	ARbReportCsvWriteStnHolding[6] := FALSE; END_IF

// Station 6
bReportCsvWriteRE_Stn[6] (CLK:=tStn6.Q OR GeneratorComparison.ARUpdate_bIntAddress[6] OR CKKTEST[7]  , Q=> );

IF bReportCsvWriteRE_Stn[6].Q THEN
	FNbCsvWriteToBuffer(
						iStationId				:=	6 , 
						sFilename				:=	sStn6tittle, 
						eCsvActionType			:=	eCsvLogData_CarrierReport , 
						udiCsvMRBCount			=> 	udiCsvMRBCount, 
						udiCsvMRBUsagePercent	=>	udiCsvMRBUsagePercent , 
						bError					=>	bErrorCsvStn[6] );
END_IF


sStn7tittle := CONCAT('_',DSLocalSystemTimeML.sCurrentDate_General);
sStn7tittle := CONCAT(DSStnBasketInfo[7].ARsBarcodeData[1],sStn7tittle);
sStn7tittle := CONCAT('-',sStn7tittle);
sStn7tittle := CONCAT(DSStnBasketInfo[7].ARsBarcodeData[2],sStn7tittle);
sStn7tittle := CONCAT('-',sStn7tittle);
sStn7tittle := CONCAT(DSStnBasketInfo[7].ARsBarcodeData[3],sStn7tittle);
sStn7tittle := CONCAT('-',sStn7tittle);
sStn7tittle := CONCAT(DSStnBasketInfo[7].sReservedInt,sStn7tittle);

ARtReportCsvWriteStnHolding[7](IN:=ARbReportCsvWriteStnHolding[7] , PT:=T#3S , Q=> , ET=> );
IF bReportCsvWriteRE_Stn[7].Q 		THEN 	ARbReportCsvWriteStnHolding[7] := TRUE; END_IF
IF ARtReportCsvWriteStnHolding[7].Q THEN	ARbReportCsvWriteStnHolding[7] := FALSE; END_IF

// Station 7
bReportCsvWriteRE_Stn[7] (CLK:=tStn7.Q OR GeneratorComparison.ARUpdate_bIntAddress[7] OR CKKTEST[8]  , Q=> );

IF  bReportCsvWriteRE_Stn[7].Q THEN
	FNbCsvWriteToBuffer(
						iStationId				:=	7 , 
						sFilename				:=	sStn7tittle, 
						eCsvActionType			:=	eCsvLogData_CarrierReport , 
						udiCsvMRBCount			=> 	udiCsvMRBCount, 
						udiCsvMRBUsagePercent	=>	udiCsvMRBUsagePercent , 
						bError					=>	bErrorCsvStn[7] );
END_IF


sStn8tittle := CONCAT('_',DSLocalSystemTimeML.sCurrentDate_General);
sStn8tittle := CONCAT(DSStnBasketInfo[8].ARsBarcodeData[1],sStn8tittle);
sStn8tittle := CONCAT('-',sStn8tittle);
sStn8tittle := CONCAT(DSStnBasketInfo[8].ARsBarcodeData[2],sStn8tittle);
sStn8tittle := CONCAT('-',sStn8tittle);
sStn8tittle := CONCAT(DSStnBasketInfo[8].ARsBarcodeData[3],sStn8tittle);
sStn8tittle := CONCAT('-',sStn8tittle);
sStn8tittle := CONCAT(DSStnBasketInfo[8].sReservedInt,sStn8tittle);

ARtReportCsvWriteStnHolding[8](IN:=ARbReportCsvWriteStnHolding[8] , PT:=T#3S , Q=> , ET=> );
IF bReportCsvWriteRE_Stn[8].Q 		THEN 	ARbReportCsvWriteStnHolding[8] := TRUE; END_IF
IF ARtReportCsvWriteStnHolding[8].Q THEN	ARbReportCsvWriteStnHolding[8] := FALSE; END_IF

// Station 8
bReportCsvWriteRE_Stn[8] (CLK:=tStn8.Q OR GeneratorComparison.ARUpdate_bIntAddress[8] OR CKKTEST[9]  , Q=> );

IF  bReportCsvWriteRE_Stn[8].Q THEN
	FNbCsvWriteToBuffer(
						iStationId				:=	8 , 
						sFilename				:=	sStn8tittle, 
						eCsvActionType			:=	eCsvLogData_CarrierReport , 
						udiCsvMRBCount			=> 	udiCsvMRBCount, 
						udiCsvMRBUsagePercent	=>	udiCsvMRBUsagePercent , 
						bError					=>	bErrorCsvStn[8] );
END_IF


sStn9tittle := CONCAT('_',DSLocalSystemTimeML.sCurrentDate_General);
sStn9tittle := CONCAT(DSStnBasketInfo[9].ARsBarcodeData[1],sStn9tittle);
sStn9tittle := CONCAT('-',sStn9tittle);
sStn9tittle := CONCAT(DSStnBasketInfo[9].ARsBarcodeData[2],sStn9tittle);
sStn9tittle := CONCAT('-',sStn9tittle);
sStn9tittle := CONCAT(DSStnBasketInfo[9].ARsBarcodeData[3],sStn9tittle);
sStn9tittle := CONCAT('-',sStn9tittle);
sStn9tittle := CONCAT(DSStnBasketInfo[9].sReservedInt,sStn9tittle);

ARtReportCsvWriteStnHolding[9](IN:=ARbReportCsvWriteStnHolding[9] , PT:=T#3S , Q=> , ET=> );
IF bReportCsvWriteRE_Stn[9].Q 		THEN 	ARbReportCsvWriteStnHolding[9] := TRUE; END_IF
IF ARtReportCsvWriteStnHolding[9].Q THEN	ARbReportCsvWriteStnHolding[9] := FALSE; END_IF

// Station 9
bReportCsvWriteRE_Stn[9] (CLK:=tStn9.Q OR CKKTEST[10]  , Q=> );

IF bReportCsvWriteRE_Stn[9].Q THEN
	FNbCsvWriteToBuffer(
						iStationId				:=	9 , 
						sFilename				:=	sStn9tittle, 
						eCsvActionType			:=	eCsvLogData_CarrierReport , 
						udiCsvMRBCount			=> 	udiCsvMRBCount, 
						udiCsvMRBUsagePercent	=>	udiCsvMRBUsagePercent , 
						bError					=>	bErrorCsvStn[9] );
END_IF


sStn10tittle := CONCAT('_',DSLocalSystemTimeML.sCurrentDate_General);
sStn10tittle := CONCAT(DSStnBasketInfo[10].ARsBarcodeData[1],sStn10tittle);
sStn10tittle := CONCAT('-',sStn10tittle);
sStn10tittle := CONCAT(DSStnBasketInfo[10].ARsBarcodeData[2],sStn10tittle);
sStn10tittle := CONCAT('-',sStn10tittle);
sStn10tittle := CONCAT(DSStnBasketInfo[10].ARsBarcodeData[3],sStn10tittle);
sStn10tittle := CONCAT('-',sStn10tittle);
sStn10tittle := CONCAT(DSStnBasketInfo[10].sReservedInt,sStn10tittle);

ARtReportCsvWriteStnHolding[10](IN:=ARbReportCsvWriteStnHolding[10] , PT:=T#3S , Q=> , ET=> );
IF bReportCsvWriteRE_Stn[10].Q 		THEN 	ARbReportCsvWriteStnHolding[10] := TRUE; END_IF
IF ARtReportCsvWriteStnHolding[10].Q THEN	ARbReportCsvWriteStnHolding[10] := FALSE; END_IF

// Station 10
bReportCsvWriteRE_Stn[10] (CLK:=tStn10.Q OR CKKTEST[11]  , Q=> );

IF bReportCsvWriteRE_Stn[10].Q THEN
	FNbCsvWriteToBuffer(
						iStationId				:=	10 , 
						sFilename				:=	sStn10tittle, 
						eCsvActionType			:=	eCsvLogData_CarrierReport , 
						udiCsvMRBCount			=> 	udiCsvMRBCount, 
						udiCsvMRBUsagePercent	=>	udiCsvMRBUsagePercent , 
						bError					=>	bErrorCsvStn[10] );
END_IF

// Station 11
//bReportCsvWriteRE_Stn[11] (CLK:=tReportCsvEn_Stn[11].Q OR CKKTEST[12]  , Q=> );
//IF (*dsMcCarrierInfo.ARStn[5].bAvailability AND*) bReportCsvWriteRE_Stn[11].Q THEN
//	FNbCsvWriteToBuffer(
//						iStationId				:=	11 , 
//						sFilename				:=	dsMcCarrierInfo.ARStn[11].sFileName, 
//						eCsvActionType			:=	eCsvLogData_CarrierReport , 
//						udiCsvMRBCount			=> 	udiCsvMRBCount, 
//						udiCsvMRBUsagePercent	=>	udiCsvMRBUsagePercent , 
//						bError					=>	bErrorCsvStn[12] );
//END_IF

// Station 12
//bReportCsvWriteRE_Stn[12] (CLK:=tReportCsvEn_Stn[12].Q OR CKKTEST[13]  , Q=> );
//IF (*dsMcCarrierInfo.ARStn[5].bAvailability AND*) bReportCsvWriteRE_Stn[12].Q THEN
//	FNbCsvWriteToBuffer(
//						iStationId				:=	12 , 
//						sFilename				:=	dsMcCarrierInfo.ARStn[12].sFileName, 
//						eCsvActionType			:=	eCsvLogData_CarrierReport , 
//						udiCsvMRBCount			=> 	udiCsvMRBCount, 
//						udiCsvMRBUsagePercent	=>	udiCsvMRBUsagePercent , 
//						bError					=>	bErrorCsvStn[12] );
//END_IF


sStn13tittle := CONCAT('_',DSLocalSystemTimeML.sCurrentDate_General);
sStn13tittle := CONCAT(AR2sDSCv_UldConfirmBasketInfo[1,1].ARsBarcodeData[1],sStn13tittle);
sStn13tittle := CONCAT('-',sStn13tittle);
sStn13tittle := CONCAT(AR2sDSCv_UldConfirmBasketInfo[1,1].ARsBarcodeData[2],sStn13tittle);
sStn13tittle := CONCAT('-',sStn13tittle);
sStn13tittle := CONCAT(AR2sDSCv_UldConfirmBasketInfo[1,1].ARsBarcodeData[3],sStn13tittle);
sStn13tittle := CONCAT('-',sStn13tittle);
sStn13tittle := CONCAT(AR2sDSCv_UldConfirmBasketInfo[1,1].sReservedInt,sStn13tittle);

tReportCsvWriteUldHolding(IN:=bReportCsvWriteUldHolding , PT:=T#3S , Q=> , ET=> );
IF bReportCsvWriteRE_Uld.Q THEN bReportCsvWriteUldHolding := TRUE; END_IF
IF tReportCsvWriteUldHolding.Q THEN	bReportCsvWriteUldHolding := FALSE; END_IF

// Unloading
bReportCsvWriteRE_Uld(CLK:=tStn13.Q OR AR2sDSCv_UldConfirmBasketInfo[1,1].bAvailibility OR CKKTEST[13]  , Q=> );

IF   bReportCsvWriteRE_Uld.Q THEN
	FNbCsvWriteToBuffer(
						iStationId				:=	81 , 
						sFilename				:=	sStn13tittle , 
						eCsvActionType			:=	eCsvGenerate_CarrierReport , 
						udiCsvMRBCount			=> 	udiCsvMRBCount, 
						udiCsvMRBUsagePercent	=>	udiCsvMRBUsagePercent , 
						bError					=>	bErrorCsvUld );
END_IF

	
fbCsvHandler(
			bEn								:=	TRUE	 , 			
			bReset							:=	bReset	 , 			
			bShutdownRequestFlag			:=	bCsvShutdownRequestFlag	 , 			
			bIdle							=>	bIdleFlag	 , 			
			bProgress						=>	bProgressFlag	 , 			
			bReadyToShutdownFlag			=>	bCsvReadyToShutdownFlag	 , 			
			bError							=>	bErrorFlag	 , 			
			bErrorCaseId					=>	iErrorCaseId	 , 			
			bClearErrorLog					:=	bClearErrorLog	 , 			
			udiCsvMRBCount					:=	udiCsvMRBCount	 , 			
			udiCsvMRBUsagePercent			:=	udiCsvMRBUsagePercent	 );

END_PROGRAM

// ---- POUs/MainProgram/DataManagement_Barcode/GeneratorComparison.TcPOU
PROGRAM GeneratorComparison
VAR
	ARbENRE 						: ARRAY[1..iUSGeneratorQty] OF R_TRIG;
	ARBufferFreqiIntAddress 			: ARRAY[1..iUSGeneratorQty] OF INT;
	ARBufferPoweriIntAddress 			: ARRAY[1..iUSGeneratorQty] OF INT;
	ARUpdate_bIntAddress 			: ARRAY[1..iUSGeneratorQty] OF BOOL;
	bTest							: BOOL;
	TON1: TON;
	TON2: TON;
	TON3: TON;
	TON4: TON;
	TON5: TON;
	TON6: TON;
	TON7: TON;
	TON8: TON;
END_VAR

;(*(*Station 1 US*)
ARbENRE[1](CLK:=bAutoStartPb OR ARbDO[eY10100_Stn01UltrasonicGeneratorOn_Off] , Q=> );
IF ARbENRE[1].Q THEN

	ARBufferFreqiIntAddress[1] := iDisplayFreqUs[1];
	ARBufferPoweriIntAddress[1] := ARDsStnSeqProcessCtrl[1].Out_DSStnSeqProOutput.i3ProTankBtmUsAPwrPercent;

END_IF

(*Program*)
TON1(IN:= bAutoStartPb AND ARbDO[eY10100_Stn01UltrasonicGeneratorOn_Off], PT:= T#10S , Q=> , ET=> );

IF TON1.Q THEN

ARUpdate_bIntAddress[1] := FALSE;

	IF (ARBufferFreqiIntAddress[1] <> iDisplayFreqUs[1]) OR (ARBufferPoweriIntAddress[1] <> ARDsStnSeqProcessCtrl[1].Out_DSStnSeqProOutput.i3ProTankBtmUsAPwrPercent) THEN
		ARUpdate_bIntAddress[1] := TRUE;
	END_IF

	IF ARUpdate_bIntAddress[1] THEN
		ARBufferFreqiIntAddress[1] := iDisplayFreqUs[1];
		ARBufferPoweriIntAddress[1] := ARDsStnSeqProcessCtrl[1].Out_DSStnSeqProOutput.i3ProTankBtmUsAPwrPercent;
	END_IF

ELSE

ARUpdate_bIntAddress[1] := FALSE;

END_IF


(*Station 2 US*)
ARbENRE[2](CLK:=bAutoStartPb OR ARbDO[eY10101_Stn02UltrasonicGeneratorOn_Off] , Q=> );
IF ARbENRE[2].Q THEN

	ARBufferFreqiIntAddress[2] := iDisplayFreqUs[2];
	ARBufferPoweriIntAddress[2] := ARDsStnSeqProcessCtrl[2].Out_DSStnSeqProOutput.i3ProTankBtmUsAPwrPercent;

END_IF

(*Program*)
TON2(IN:= bAutoStartPb AND ARbDO[eY10101_Stn02UltrasonicGeneratorOn_Off], PT:= T#10S , Q=> , ET=> );

IF TON2.Q THEN

ARUpdate_bIntAddress[2] := FALSE;

	IF (ARBufferFreqiIntAddress[2] <> iDisplayFreqUs[2]) OR (ARBufferPoweriIntAddress[2] <> ARDsStnSeqProcessCtrl[2].Out_DSStnSeqProOutput.i3ProTankBtmUsAPwrPercent) THEN
		ARUpdate_bIntAddress[2] := TRUE;
	END_IF

	IF ARUpdate_bIntAddress[2] THEN
		ARBufferFreqiIntAddress[2] := iDisplayFreqUs[2];
		ARBufferPoweriIntAddress[2] := ARDsStnSeqProcessCtrl[2].Out_DSStnSeqProOutput.i3ProTankBtmUsAPwrPercent;
	END_IF

ELSE

ARUpdate_bIntAddress[2] := FALSE;

END_IF


(*Station 3 US*)
ARbENRE[3](CLK:=bAutoStartPb OR ARbDO[eY11100_Stn03MegasonicGenerator01On_Off] OR ARbDO[eY11101_Stn03MegasonicGenerator02On_Off] , Q=> );
IF ARbENRE[3].Q THEN

	//ARBufferFreqiIntAddress[3] := iDisplayFreqUs[3];
	ARBufferPoweriIntAddress[3] := ARDsStnSeqProcessCtrl[3].Out_DSStnSeqProOutput.i3ProTankBtmUsAPwrPercent;

END_IF

(*Program*)
TON3(IN:= bAutoStartPb AND (ARbDO[eY11100_Stn03MegasonicGenerator01On_Off] OR ARbDO[eY11101_Stn03MegasonicGenerator02On_Off]), PT:= T#10S , Q=> , ET=> );

IF TON3.Q THEN

ARUpdate_bIntAddress[3] := FALSE;

	IF (*(ARBufferFreqiIntAddress[3] <> DSWeberEnclosure[1].DSWeberGenerator[3].IN_iFreqSetPoint) OR*) (ARBufferPoweriIntAddress[3] <> ARDsStnSeqProcessCtrl[3].Out_DSStnSeqProOutput.i3ProTankBtmUsAPwrPercent) THEN
		ARUpdate_bIntAddress[3] := TRUE;
	END_IF

	IF ARUpdate_bIntAddress[3] THEN
	//	ARBufferFreqiIntAddress[3] := DSWeberEnclosure[1].DSWeberGenerator[3].IN_iFreqSetPoint;
		ARBufferPoweriIntAddress[3] := ARDsStnSeqProcessCtrl[3].Out_DSStnSeqProOutput.i3ProTankBtmUsAPwrPercent;
	END_IF

ELSE

ARUpdate_bIntAddress[3] := FALSE;

END_IF


(*Station 4 US*)
ARbENRE[4](CLK:=bAutoStartPb OR ARbDO[eY10102_Stn04UltrasonicGeneratorOn_Off] , Q=> );
IF ARbENRE[4].Q THEN

	ARBufferFreqiIntAddress[4] := iDisplayFreqUs[4];
	ARBufferPoweriIntAddress[4] := ARDsStnSeqProcessCtrl[4].Out_DSStnSeqProOutput.i3ProTankBtmUsAPwrPercent;

END_IF

(*Program*)
TON4(IN:= bAutoStartPb AND ARbDO[eY10102_Stn04UltrasonicGeneratorOn_Off], PT:= T#10S , Q=> , ET=> );

IF TON4.Q THEN

ARUpdate_bIntAddress[4] := FALSE;

	IF (ARBufferFreqiIntAddress[4] <> iDisplayFreqUs[4]) OR (ARBufferPoweriIntAddress[4] <> ARDsStnSeqProcessCtrl[4].Out_DSStnSeqProOutput.i3ProTankBtmUsAPwrPercent) THEN
		ARUpdate_bIntAddress[4] := TRUE;
	END_IF

	IF ARUpdate_bIntAddress[4] THEN
		ARBufferFreqiIntAddress[4] := iDisplayFreqUs[4];
		ARBufferPoweriIntAddress[4] := ARDsStnSeqProcessCtrl[4].Out_DSStnSeqProOutput.i3ProTankBtmUsAPwrPercent;
	END_IF

ELSE

ARUpdate_bIntAddress[4] := FALSE;

END_IF


(*Station 5 US*)
ARbENRE[5](CLK:=bAutoStartPb OR ARbDO[eY10103_Stn05UltrasonicGeneratorOn_Off] , Q=> );
IF ARbENRE[5].Q THEN

	ARBufferFreqiIntAddress[5] := iDisplayFreqUs[5];
	ARBufferPoweriIntAddress[5] := ARDsStnSeqProcessCtrl[5].Out_DSStnSeqProOutput.i3ProTankBtmUsAPwrPercent;

END_IF

(*Program*)
TON5(IN:= bAutoStartPb AND ARbDO[eY10103_Stn05UltrasonicGeneratorOn_Off], PT:= T#10S , Q=> , ET=> );

IF TON5.Q THEN

ARUpdate_bIntAddress[5] := FALSE;

	IF (ARBufferFreqiIntAddress[5] <> iDisplayFreqUs[5]) OR (ARBufferPoweriIntAddress[5] <> ARDsStnSeqProcessCtrl[5].Out_DSStnSeqProOutput.i3ProTankBtmUsAPwrPercent) THEN
		ARUpdate_bIntAddress[5] := TRUE;
	END_IF

	IF ARUpdate_bIntAddress[5] THEN
		ARBufferFreqiIntAddress[5] := iDisplayFreqUs[5];
		ARBufferPoweriIntAddress[5] := ARDsStnSeqProcessCtrl[5].Out_DSStnSeqProOutput.i3ProTankBtmUsAPwrPercent;
	END_IF

ELSE

ARUpdate_bIntAddress[5] := FALSE;

END_IF


(*Station 6 US*)
ARbENRE[6](CLK:=bAutoStartPb OR ARbDO[eY12001_Stn06MegasonicGenerator01On_Off] OR ARbDO[eY12002_Stn06MegasonicGenerator02On_Off] OR ARbDO[eY12003_Stn06MegasonicGenerator03On_Off] , Q=> );
IF ARbENRE[6].Q THEN

	//ARBufferFreqiIntAddress[6] := iDisplayFreqUs[6];
	ARBufferPoweriIntAddress[6] := ARDsStnSeqProcessCtrl[6].Out_DSStnSeqProOutput.i3ProTankBtmUsAPwrPercent;

END_IF

(*Program*)
TON6(IN:= bAutoStartPb AND (ARbDO[eY12001_Stn06MegasonicGenerator01On_Off] OR ARbDO[eY12002_Stn06MegasonicGenerator02On_Off] OR ARbDO[eY12003_Stn06MegasonicGenerator03On_Off]), PT:= T#10S , Q=> , ET=> );

IF TON6.Q THEN

ARUpdate_bIntAddress[6] := FALSE;

	IF (*(ARBufferFreqiIntAddress[6] <> DSWeberEnclosure[1].DSWeberGenerator[6].IN_iFreqSetPoint) OR*) (ARBufferPoweriIntAddress[6] <> ARDsStnSeqProcessCtrl[6].Out_DSStnSeqProOutput.i3ProTankBtmUsAPwrPercent) THEN
		ARUpdate_bIntAddress[6] := TRUE;
	END_IF

	IF ARUpdate_bIntAddress[6] THEN
	//	ARBufferFreqiIntAddress[6] := DSWeberEnclosure[1].DSWeberGenerator[6].IN_iFreqSetPoint;
		ARBufferPoweriIntAddress[6] := ARDsStnSeqProcessCtrl[6].Out_DSStnSeqProOutput.i3ProTankBtmUsAPwrPercent;
	END_IF

ELSE

ARUpdate_bIntAddress[6] := FALSE;

END_IF


(*Station 7 US*)
ARbENRE[7](CLK:=bAutoStartPb OR ARbDO[eY10104_Stn07UltrasonicGeneratorOn_Off] , Q=> );
IF ARbENRE[7].Q THEN

	ARBufferFreqiIntAddress[7] := iDisplayFreqUs[7];
	ARBufferPoweriIntAddress[7] := ARDsStnSeqProcessCtrl[7].Out_DSStnSeqProOutput.i3ProTankBtmUsAPwrPercent;

END_IF

(*Program*)
TON7(IN:= bAutoStartPb AND ARbDO[eY10104_Stn07UltrasonicGeneratorOn_Off], PT:= T#10S , Q=> , ET=> );

IF TON7.Q THEN

ARUpdate_bIntAddress[7] := FALSE;

	IF (ARBufferFreqiIntAddress[7] <> iDisplayFreqUs[7]) OR (ARBufferPoweriIntAddress[7] <> ARDsStnSeqProcessCtrl[7].Out_DSStnSeqProOutput.i3ProTankBtmUsAPwrPercent) THEN
		ARUpdate_bIntAddress[7] := TRUE;
	END_IF

	IF ARUpdate_bIntAddress[7] THEN
		ARBufferFreqiIntAddress[7] := iDisplayFreqUs[7];
		ARBufferPoweriIntAddress[7] := ARDsStnSeqProcessCtrl[7].Out_DSStnSeqProOutput.i3ProTankBtmUsAPwrPercent;
	END_IF

ELSE

ARUpdate_bIntAddress[7] := FALSE;

END_IF


(*Station 8 US*)
ARbENRE[8](CLK:=bAutoStartPb OR ARbDO[eY10105_Stn08UltrasonicGeneratorOn_Off] , Q=> );
IF ARbENRE[8].Q THEN

	ARBufferFreqiIntAddress[8] := iDisplayFreqUs[8];
	ARBufferPoweriIntAddress[8] := ARDsStnSeqProcessCtrl[8].Out_DSStnSeqProOutput.i3ProTankBtmUsAPwrPercent;

END_IF

(*Program*)
TON8(IN:= bAutoStartPb AND ARbDO[eY10105_Stn08UltrasonicGeneratorOn_Off], PT:= T#10S , Q=> , ET=> );

IF TON8.Q THEN

ARUpdate_bIntAddress[8] := FALSE;

	IF (ARBufferFreqiIntAddress[8] <> iDisplayFreqUs[8]) OR (ARBufferPoweriIntAddress[8] <> ARDsStnSeqProcessCtrl[8].Out_DSStnSeqProOutput.i3ProTankBtmUsAPwrPercent) THEN
		ARUpdate_bIntAddress[8] := TRUE;
	END_IF

	IF ARUpdate_bIntAddress[8] THEN
		ARBufferFreqiIntAddress[8] := iDisplayFreqUs[8];
		ARBufferPoweriIntAddress[8] := ARDsStnSeqProcessCtrl[8].Out_DSStnSeqProOutput.i3ProTankBtmUsAPwrPercent;
	END_IF

ELSE

ARUpdate_bIntAddress[8] := FALSE;

END_IF
*)

END_PROGRAM

// ---- POUs/MainProgram/Csv/Csv_Report_Mapping.TcPOU
PROGRAM Csv_Report_Mapping
VAR
	sTime: STRING(20);
	
	
END_VAR

	sTime  		:= CONCAT(DSLocalSystemTimeML.s12Hour, ':');
	sTime  		:= CONCAT(sTime, DSLocalSystemTimeML.sMin);
//	sTime  		:= CONCAT(sTime, ':');
//	sTime  		:= CONCAT(sTime, DSLocalSystemTimeML.sSec);
	sTime  		:= CONCAT(sTime, ' ');
	sTime 		:= CONCAT(sTime, DSLocalSystemTimeML.s12HrSign);

// Configure total report to log
dsCsvReport.iNumOfData_HeadlineData		:= 30;
dsCsvReport.iNumOfData_HeadlineTitle	:= 30;
dsCsvReport.iNumOfData_LogData			:= 45;
dsCsvReport.iNumOfData_LogTitle			:= 45;
dsCsvReport.iNumOfData_LogUnit			:= 45;

// Headline Title ( FIRST ROW )
dsCsvReport.ARsHeadlineTitle[1]  := '';
dsCsvReport.ARsHeadlineTitle[2]  := 'Operator';
dsCsvReport.ARsHeadlineTitle[3]  := 'Loading ID';
dsCsvReport.ARsHeadlineTitle[4]  := 'Unloading ID';
dsCsvReport.ARsHeadlineTitle[5]  := 'Product Recipe Number';
dsCsvReport.ARsHeadlineTitle[6]  := 'Product Recipe Description';
dsCsvReport.ARsHeadlineTitle[7]  := 'Load Number';
dsCsvReport.ARsHeadlineTitle[8]  := '';
dsCsvReport.ARsHeadlineTitle[9]  := '';
dsCsvReport.ARsHeadlineTitle[10] := '';
dsCsvReport.ARsHeadlineTitle[11] := '';
dsCsvReport.ARsHeadlineTitle[12] := '';
dsCsvReport.ARsHeadlineTitle[13] := '';
dsCsvReport.ARsHeadlineTitle[14] := '';
dsCsvReport.ARsHeadlineTitle[15] := '';


// Headline Data ( SECOND ROW )
dsCsvReport.ARsHeadlineData[1]  := '';
dsCsvReport.ARsHeadlineData[2]  := fbHmiTF1800_UserlevelManagement.dsHmiUserStatus_Active.sLoginName;
dsCsvReport.ARsHeadlineData[3]  := '1';
dsCsvReport.ARsHeadlineData[4]  := '1';
dsCsvReport.ARsHeadlineData[5]  := INT_TO_STRING(AR2sDSCv_LdConfirmBasketInfo[1,4].iProductRecipeNo);
dsCsvReport.ARsHeadlineData[6]  := AR2sDSCv_LdConfirmBasketInfo[1,4].sProgramDescription;
dsCsvReport.ARsHeadlineData[7]  := INT_TO_STRING(iProgBatchTotal);
dsCsvReport.ARsHeadlineData[8]  := '';
dsCsvReport.ARsHeadlineData[9]  := '';
dsCsvReport.ARsHeadlineData[10] := '';
dsCsvReport.ARsHeadlineData[11] := '';
dsCsvReport.ARsHeadlineData[12] := '';
dsCsvReport.ARsHeadlineData[13] := '';
dsCsvReport.ARsHeadlineData[14] := '';
dsCsvReport.ARsHeadlineData[15] := '';

// Data log unit ( THIRD ROW )
dsCsvReport.ARsLogUnit[1]:='';   
dsCsvReport.ARsLogUnit[2]:='N/A';
dsCsvReport.ARsLogUnit[3]:='N/A';
dsCsvReport.ARsLogUnit[4]:='N/A';
dsCsvReport.ARsLogUnit[5]:='N/A';
dsCsvReport.ARsLogUnit[6]:='N/A';
dsCsvReport.ARsLogUnit[7]:='N/A';
dsCsvReport.ARsLogUnit[8]:='Sec';
dsCsvReport.ARsLogUnit[9]:='Sec';
dsCsvReport.ARsLogUnit[10]:='Sec'; 
dsCsvReport.ARsLogUnit[11]:='Sec'; 
dsCsvReport.ARsLogUnit[12]:='Sec'; 
dsCsvReport.ARsLogUnit[13]:='Sec'; 
dsCsvReport.ARsLogUnit[14]:='DegC';
dsCsvReport.ARsLogUnit[15]:='DegC';
dsCsvReport.ARsLogUnit[16]:='%';   
dsCsvReport.ARsLogUnit[17]:='%';   
dsCsvReport.ARsLogUnit[18]:='Hz';  
dsCsvReport.ARsLogUnit[19]:='Hz';  
dsCsvReport.ARsLogUnit[20]:='%';   
dsCsvReport.ARsLogUnit[21]:='%';   
dsCsvReport.ARsLogUnit[22]:='Hz';  
dsCsvReport.ARsLogUnit[23]:='Hz';  
dsCsvReport.ARsLogUnit[24]:='%';   
dsCsvReport.ARsLogUnit[25]:='%';   
dsCsvReport.ARsLogUnit[26]:='Hz';  
dsCsvReport.ARsLogUnit[27]:='Hz';  
dsCsvReport.ARsLogUnit[28]:='%';   
dsCsvReport.ARsLogUnit[29]:='%';   
dsCsvReport.ARsLogUnit[30]:='Hz';  
dsCsvReport.ARsLogUnit[31]:='Hz';  
dsCsvReport.ARsLogUnit[32]:='Kpa'; 
dsCsvReport.ARsLogUnit[33]:='Kpa'; 
dsCsvReport.ARsLogUnit[34]:='uS';  
dsCsvReport.ARsLogUnit[35]:='uS';  
dsCsvReport.ARsLogUnit[36]:='LPM'; 
dsCsvReport.ARsLogUnit[37]:='LPM'; 
dsCsvReport.ARsLogUnit[38]:='OHM'; 
dsCsvReport.ARsLogUnit[39]:='OHM'; 
dsCsvReport.ARsLogUnit[40]:='PH';  
dsCsvReport.ARsLogUnit[41]:='PH';  
dsCsvReport.ARsLogUnit[42]:='N/A'; 
dsCsvReport.ARsLogUnit[43]:='N/A'; 
dsCsvReport.ARsLogUnit[44]:='Sec'; 
dsCsvReport.ARsLogUnit[45]:='Sec'; 

// Data log unit ( FORTH ROW )
dsCsvReport.ARsLogTitle[1]:='Time';
dsCsvReport.ARsLogTitle[2]:='Station';         
dsCsvReport.ARsLogTitle[3]:='Station';         
dsCsvReport.ARsLogTitle[4]:='Sequences Recipe';
dsCsvReport.ARsLogTitle[5]:='Sequences Recipe';
dsCsvReport.ARsLogTitle[6]:='Sub Recipe';      
dsCsvReport.ARsLogTitle[7]:='Sub Recipe';      
dsCsvReport.ARsLogTitle[8]:='Minimum Time';    
dsCsvReport.ARsLogTitle[9]:='Minimum Time';    
dsCsvReport.ARsLogTitle[10]:='Maximum Time';    
dsCsvReport.ARsLogTitle[11]:='Maximum Time';              
dsCsvReport.ARsLogTitle[12]:='Effective Time';            
dsCsvReport.ARsLogTitle[13]:='Effective Time';            
dsCsvReport.ARsLogTitle[14]:='Temperature';               
dsCsvReport.ARsLogTitle[15]:='Temperature';               
dsCsvReport.ARsLogTitle[16]:='U/Sonic Bottom A Power';    
dsCsvReport.ARsLogTitle[17]:='U/Sonic Bottom A Power';    
dsCsvReport.ARsLogTitle[18]:='U/Sonic Bottom A Frequency';
dsCsvReport.ARsLogTitle[19]:='U/Sonic Bottom A Frequency';
dsCsvReport.ARsLogTitle[20]:='U/Sonic Bottom B Power';    
dsCsvReport.ARsLogTitle[21]:='U/Sonic Bottom B Power';    
dsCsvReport.ARsLogTitle[22]:='U/Sonic Bottom B Frequency';
dsCsvReport.ARsLogTitle[23]:='U/Sonic Bottom B Frequency';
dsCsvReport.ARsLogTitle[24]:='U/Sonic Side A Power SV';   
dsCsvReport.ARsLogTitle[25]:='U/Sonic Side A Power PV';   
dsCsvReport.ARsLogTitle[26]:='U/Sonic Side A Frequency';  
dsCsvReport.ARsLogTitle[27]:='U/Sonic Side A Frequency';  
dsCsvReport.ARsLogTitle[28]:='U/Sonic Side B Power';      
dsCsvReport.ARsLogTitle[29]:='U/Sonic Side B Power';      
dsCsvReport.ARsLogTitle[30]:='U/Sonic Side B Frequency';  
dsCsvReport.ARsLogTitle[31]:='U/Sonic Side B Frequency';  
dsCsvReport.ARsLogTitle[32]:='Vacuum SV';                 
dsCsvReport.ARsLogTitle[33]:='Vacuum PV';                 
dsCsvReport.ARsLogTitle[34]:='Conductivity';              
dsCsvReport.ARsLogTitle[35]:='Conductivity';              
dsCsvReport.ARsLogTitle[36]:='Pump Flow';                 
dsCsvReport.ARsLogTitle[37]:='Pump Flow';                 
dsCsvReport.ARsLogTitle[38]:='Resistivity';               
dsCsvReport.ARsLogTitle[39]:='Resistivity';               
dsCsvReport.ARsLogTitle[40]:='PH PV';                     
dsCsvReport.ARsLogTitle[41]:='PH PV';                     
dsCsvReport.ARsLogTitle[42]:='Quality';                   
dsCsvReport.ARsLogTitle[43]:='Quality';                   
dsCsvReport.ARsLogTitle[44]:='Actual Time';               
dsCsvReport.ARsLogTitle[45]:='Actual Time';               

// Data log info STN 01 ( FIFTH ROW )
dsCsvReport.AR2sLogData[1][1]:=sTime;
dsCsvReport.AR2sLogData[1][2]:='N/A';(*Station*)                                                                
dsCsvReport.AR2sLogData[1][3]:='1-SONIC CLEANING';(*Station*)                                                      
dsCsvReport.AR2sLogData[1][4]:='N/A';(*Sequences Recipe*)                                                       
dsCsvReport.AR2sLogData[1][5]:=DSHmiStationDisplayInfo[1].sStationSequenceRecipeDescription;(*Sequences Recipe*)
dsCsvReport.AR2sLogData[1][6]:='N/A';(*Sub Recipe*)                                                             
dsCsvReport.AR2sLogData[1][7]:=DSHmiStationDisplayInfo[1].sStationSubDescription;(*Sub Recipe*)                 
dsCsvReport.AR2sLogData[1][8]:=INT_TO_STRING(ARDsStnMinMaxEffTimeDisplay[1].iMinTime);(*Minimum Time*)          
dsCsvReport.AR2sLogData[1][9]:='N/A';(*Minimum Time*)                                                           
dsCsvReport.AR2sLogData[1][10]:=INT_TO_STRING(ARDsStnMinMaxEffTimeDisplay[1].iMaxTime);(*Maximum Time*)          
dsCsvReport.AR2sLogData[1][11]:='N/A';(*Maximum Time*)                                                                                   
dsCsvReport.AR2sLogData[1][12]:=INT_TO_STRING(ARDsStnMinMaxEffTimeDisplay[1].iEffTime);(*Effective Time*)                                
dsCsvReport.AR2sLogData[1][13]:='N/A';(*Effective Time*)                                                                                 
dsCsvReport.AR2sLogData[1][14]:=REAL_TO_STRING(ARrStnTempSV[1]);(*Temperature SV*)                                                       
dsCsvReport.AR2sLogData[1][15]:=REAL_TO_STRING(ARrStnTempPV[1]);(*Temperature PV*)                                                       
dsCsvReport.AR2sLogData[1][16]:=INT_TO_STRING(ARDsStnSeqProcessCtrl[1].Out_DSStnSeqProOutput.i3ProTankBtmUsAPwrPercent);(*U/Sonic Bottom A Power SV*)                                     
dsCsvReport.AR2sLogData[1][17]:=INT_TO_STRING(ARiUsPowerPV_percent[1]);(*U/Sonic Bottom A Power PV*)                                           
dsCsvReport.AR2sLogData[1][18]:='N/A';(*U/Sonic Bottom A Frequency SV*)                                                                  
dsCsvReport.AR2sLogData[1][19]:=INT_TO_STRING(iDisplayFreqUs[1]);(*U/Sonic Bottom A Frequency PV*)
dsCsvReport.AR2sLogData[1][20]:='N/A';(*U/Sonic Bottom B Power SV*)                                     
dsCsvReport.AR2sLogData[1][21]:='N/A';(*U/Sonic Bottom B Power PV*)                                           
dsCsvReport.AR2sLogData[1][22]:='N/A';(*U/Sonic Bottom B Frequency SV*)                                                                  
dsCsvReport.AR2sLogData[1][23]:='N/A';(*U/Sonic Bottom B Frequency PV*)                                                                  
dsCsvReport.AR2sLogData[1][24]:='N/A';(*U/Sonic Side A Power SV*)                                                                        
dsCsvReport.AR2sLogData[1][25]:='N/A';(*U/Sonic Side A Power PV*)                                                                        
dsCsvReport.AR2sLogData[1][26]:='N/A';(*U/Sonic Side A Frequency SV*)                                                                    
dsCsvReport.AR2sLogData[1][27]:='N/A';(*U/Sonic Side A Frequency PV*)                                                                    
dsCsvReport.AR2sLogData[1][28]:='N/A';(*U/Sonic Side B Power SV*)                                                                        
dsCsvReport.AR2sLogData[1][29]:='N/A';(*U/Sonic Side B Power PV*)                                                                        
dsCsvReport.AR2sLogData[1][30]:='N/A';(*U/Sonic Side B Frequency SV*)                                                                    
dsCsvReport.AR2sLogData[1][31]:='N/A';(*U/Sonic Side B Frequency PV*)                                                                    
dsCsvReport.AR2sLogData[1][32]:='N/A';(*Vacuum SV*)                                                                                      
dsCsvReport.AR2sLogData[1][33]:='N/A';(*Vacuum PV*)                                                                                      
dsCsvReport.AR2sLogData[1][34]:='N/A';(*Conductivity SV*)                                                                                
dsCsvReport.AR2sLogData[1][35]:=REAL_TO_STRING(ARrStnConductivityPV[1]);(*Conductivity PV*)                                              
dsCsvReport.AR2sLogData[1][36]:='N/A';(*Pump Flow SV*)                                                                                   
dsCsvReport.AR2sLogData[1][37]:=REAL_TO_STRING(ARrStnFilterPressurePV[1]);(*Pump Flow PV*)                                               
dsCsvReport.AR2sLogData[1][38]:='N/A';(*Resistivity SV*)                                                                                 
dsCsvReport.AR2sLogData[1][39]:='N/A';(*Resistivity PV*)                                                                                 
dsCsvReport.AR2sLogData[1][40]:='N/A';(*PH SV*)                                                                                          
dsCsvReport.AR2sLogData[1][41]:='N/A'; (*PH PV*)                                                                                         
dsCsvReport.AR2sLogData[1][42]:='N/A';(*Quality*)                                                                                        
dsCsvReport.AR2sLogData[1][43]:=DSStnBasketInfo[1].sProductQuality;(*Quality*)                                                           
dsCsvReport.AR2sLogData[1][44]:=INT_TO_STRING(ARDsStnSeqProcessCtrl[1].Out_iCurrentProcessTime);(*Actual Time*)                          
dsCsvReport.AR2sLogData[1][45]:='N/A';(*Actual Time*)        
                                                                            
// Data log info STN 02 ( SIX ROW )
dsCsvReport.AR2sLogData[2][1]:=sTime;(*Station*)
dsCsvReport.AR2sLogData[2][2]:='N/A';(*Station*)
dsCsvReport.AR2sLogData[2][3]:='2-RINSING';(*Station*)
dsCsvReport.AR2sLogData[2][4]:='N/A';(*Sequences Recipe*)
dsCsvReport.AR2sLogData[2][5]:=DSHmiStationDisplayInfo[2].sStationSequenceRecipeDescription;(*Sequences Recipe*)
dsCsvReport.AR2sLogData[2][6]:='N/A';(*Sub Recipe*)
dsCsvReport.AR2sLogData[2][7]:=DSHmiStationDisplayInfo[2].sStationSubDescription;(*Sub Recipe*)
dsCsvReport.AR2sLogData[2][8]:=INT_TO_STRING(ARDsStnMinMaxEffTimeDisplay[2].iMinTime);(*Minimum Time*)
dsCsvReport.AR2sLogData[2][9]:='N/A';(*Minimum Time*)
dsCsvReport.AR2sLogData[2][10]:=INT_TO_STRING(ARDsStnMinMaxEffTimeDisplay[2].iMaxTime);(*Maximum Time*)
dsCsvReport.AR2sLogData[2][11]:='N/A';(*Maximum Time*)
dsCsvReport.AR2sLogData[2][12]:=INT_TO_STRING(ARDsStnMinMaxEffTimeDisplay[2].iEffTime);(*Effective Time*)
dsCsvReport.AR2sLogData[2][13]:='N/A';(*Effective Time*)
dsCsvReport.AR2sLogData[2][14]:=REAL_TO_STRING(ARrStnTempSV[2]);(*Temperature SV*)
dsCsvReport.AR2sLogData[2][15]:=REAL_TO_STRING(ARrStnTempPV[2]);(*Temperature PV*)
dsCsvReport.AR2sLogData[2][16]:=INT_TO_STRING(ARDsStnSeqProcessCtrl[2].Out_DSStnSeqProOutput.i3ProTankBtmUsAPwrPercent);(*U/Sonic Bottom A Power SV*)
dsCsvReport.AR2sLogData[2][17]:=INT_TO_STRING(ARiUsPowerPV_percent[2]);(*U/Sonic Bottom A Power PV*)
dsCsvReport.AR2sLogData[2][18]:='N/A';(*U/Sonic Bottom A Frequency SV*)
dsCsvReport.AR2sLogData[2][19]:=INT_TO_STRING(iDisplayFreqUs[2]);(*U/Sonic Bottom A Frequency PV*)
dsCsvReport.AR2sLogData[2][20]:='N/A';(*U/Sonic Bottom B Power SV*)
dsCsvReport.AR2sLogData[2][21]:='N/A';(*U/Sonic Bottom B Power PV*)
dsCsvReport.AR2sLogData[2][22]:='N/A';(*U/Sonic Bottom B Frequency SV*)
dsCsvReport.AR2sLogData[2][23]:='N/A';(*U/Sonic Bottom B Frequency PV*)
dsCsvReport.AR2sLogData[2][24]:='N/A';(*U/Sonic Side A Power SV*)
dsCsvReport.AR2sLogData[2][25]:='N/A';(*U/Sonic Side A Power PV*)
dsCsvReport.AR2sLogData[2][26]:='N/A';(*U/Sonic Side A Frequency SV*)
dsCsvReport.AR2sLogData[2][27]:='N/A';(*U/Sonic Side A Frequency PV*)
dsCsvReport.AR2sLogData[2][28]:='N/A';(*U/Sonic Side B Power SV*)
dsCsvReport.AR2sLogData[2][29]:='N/A';(*U/Sonic Side B Power PV*)
dsCsvReport.AR2sLogData[2][30]:='N/A';(*U/Sonic Side B Frequency SV*)
dsCsvReport.AR2sLogData[2][31]:='N/A';(*U/Sonic Side B Frequency PV*)
dsCsvReport.AR2sLogData[2][32]:='N/A';(*Vacuum SV*)
dsCsvReport.AR2sLogData[2][33]:='N/A';(*Vacuum PV*)
dsCsvReport.AR2sLogData[2][34]:='N/A';(*Conductivity SV*)
dsCsvReport.AR2sLogData[2][35]:=REAL_TO_STRING(ARrStnConductivityPV[2]);(*Conductivity PV*)
dsCsvReport.AR2sLogData[2][36]:='N/A';(*Pump Flow SV*)
dsCsvReport.AR2sLogData[2][37]:=REAL_TO_STRING(ARrStnFilterPressurePV[2]);(*Pump Flow PV*)
dsCsvReport.AR2sLogData[2][38]:='N/A';(*Resistivity SV*)
dsCsvReport.AR2sLogData[2][39]:='N/A';(*Resistivity PV*)
dsCsvReport.AR2sLogData[2][40]:='N/A';(*PH SV*)
dsCsvReport.AR2sLogData[2][41]:='N/A'; (*PH PV*)
dsCsvReport.AR2sLogData[2][42]:='N/A';(*Quality*)
dsCsvReport.AR2sLogData[2][43]:=DSStnBasketInfo[2].sProductQuality;(*Quality*)
dsCsvReport.AR2sLogData[2][44]:=INT_TO_STRING(ARDsStnSeqProcessCtrl[2].Out_iCurrentProcessTime);(*Actual Time*)
dsCsvReport.AR2sLogData[2][45]:='N/A';(*Actual Time*)                 


// Data log info STN 03 ( SEVEN ROW )
dsCsvReport.AR2sLogData[3][1]  :=sTime;(*Station*)
dsCsvReport.AR2sLogData[3][2]  :='N/A';(*Station*)
dsCsvReport.AR2sLogData[3][3]  :='3-SONIC CLEANING';(*Station*)
dsCsvReport.AR2sLogData[3][4]  :='N/A';(*Sequences Recipe*)
dsCsvReport.AR2sLogData[3][5]  :=DSHmiStationDisplayInfo[3].sStationSequenceRecipeDescription;(*Sequences Recipe*)
dsCsvReport.AR2sLogData[3][6]  :='N/A';(*Sub Recipe*)
dsCsvReport.AR2sLogData[3][7]  :=DSHmiStationDisplayInfo[3].sStationSubDescription;(*Sub Recipe*)
dsCsvReport.AR2sLogData[3][8]  :=INT_TO_STRING(ARDsStnMinMaxEffTimeDisplay[3].iMinTime);(*Minimum Time*)
dsCsvReport.AR2sLogData[3][9]  :='N/A';(*Minimum Time*)
dsCsvReport.AR2sLogData[3][10]  :=INT_TO_STRING(ARDsStnMinMaxEffTimeDisplay[3].iMaxTime);(*Maximum Time*)
dsCsvReport.AR2sLogData[3][11] :='N/A';(*Maximum Time*)
dsCsvReport.AR2sLogData[3][12] :=INT_TO_STRING(ARDsStnMinMaxEffTimeDisplay[3].iEffTime);(*Effective Time*)
dsCsvReport.AR2sLogData[3][13] :='N/A';(*Effective Time*)
dsCsvReport.AR2sLogData[3][14] :=REAL_TO_STRING(ARrStnTempSV[3]);(*Temperature SV*)
dsCsvReport.AR2sLogData[3][15] :=REAL_TO_STRING(ARrStnTempPV[3]);(*Temperature PV*)
dsCsvReport.AR2sLogData[3][16] :=INT_TO_STRING(ARDsStnSeqProcessCtrl[3].Out_DSStnSeqProOutput.i3ProTankBtmUsAPwrPercent);(*U/Sonic Bottom A Power SV*)
dsCsvReport.AR2sLogData[3][17]:=INT_TO_STRING(ARiMegaPowerPV_percent[1]);(*U/Sonic Bottom A Power PV*)
dsCsvReport.AR2sLogData[3][18]:='N/A';(*U/Sonic Bottom A Frequency SV*)
dsCsvReport.AR2sLogData[3][19]:=INT_TO_STRING(DSV2ModbusControl2.wModbusData[1]);(*U/Sonic Bottom A Frequency PV*)
dsCsvReport.AR2sLogData[3][20]:='N/A';(*U/Sonic Bottom B Power SV*)
dsCsvReport.AR2sLogData[3][21]:='N/A';(*U/Sonic Bottom B Power PV*)
dsCsvReport.AR2sLogData[3][22]:='N/A';(*U/Sonic Bottom B Frequency SV*)
dsCsvReport.AR2sLogData[3][23]:='N/A';(*U/Sonic Bottom B Frequency PV*)
dsCsvReport.AR2sLogData[3][24]:='N/A';(*U/Sonic Side A Power SV*)
dsCsvReport.AR2sLogData[3][25]:='N/A';(*U/Sonic Side A Power PV*)
dsCsvReport.AR2sLogData[3][26]:='N/A';(*U/Sonic Side A Frequency SV*)
dsCsvReport.AR2sLogData[3][27]:='N/A';(*U/Sonic Side A Frequency PV*)
dsCsvReport.AR2sLogData[3][28]:='N/A';(*U/Sonic Side B Power SV*)
dsCsvReport.AR2sLogData[3][29]:='N/A';(*U/Sonic Side B Power PV*)
dsCsvReport.AR2sLogData[3][30]:='N/A';(*U/Sonic Side B Frequency SV*)
dsCsvReport.AR2sLogData[3][31]:='N/A';(*U/Sonic Side B Frequency PV*)
dsCsvReport.AR2sLogData[3][32]:='N/A';(*Vacuum SV*)
dsCsvReport.AR2sLogData[3][33]:='N/A';(*Vacuum PV*)
dsCsvReport.AR2sLogData[3][34]:='N/A';(*Conductivity SV*)
dsCsvReport.AR2sLogData[3][35]:=REAL_TO_STRING(ARrStnConductivityPV[3]);(*Conductivity PV*)
dsCsvReport.AR2sLogData[3][36]:='N/A';(*Pump Flow SV*)
dsCsvReport.AR2sLogData[3][37]:=REAL_TO_STRING(ARrStnFilterPressurePV[3]);(*Pump Flow PV*)
dsCsvReport.AR2sLogData[3][38]:='N/A';(*Resistivity SV*)
dsCsvReport.AR2sLogData[3][39]:='N/A';(*Resistivity PV*)
dsCsvReport.AR2sLogData[3][40]:='N/A';(*PH SV*)
dsCsvReport.AR2sLogData[3][41]:='N/A'; (*PH PV*)
dsCsvReport.AR2sLogData[3][42]:='N/A';(*Quality*)
dsCsvReport.AR2sLogData[3][43]:=DSStnBasketInfo[3].sProductQuality;(*Quality*)
dsCsvReport.AR2sLogData[3][44]:=INT_TO_STRING(ARDsStnSeqProcessCtrl[3].Out_iCurrentProcessTime);(*Actual Time*)
dsCsvReport.AR2sLogData[3][45]:='N/A';(*Actual Time*)                                        

// Data log info STN 04 ( EIGHT ROW )4-RINSING
dsCsvReport.AR2sLogData[4][1]  :=sTime;
dsCsvReport.AR2sLogData[4][2]  :='N/A';(*Station*)
dsCsvReport.AR2sLogData[4][3]  :='4-RINSING';(*Station*)
dsCsvReport.AR2sLogData[4][4]  :='N/A';(*Sequences Recipe*)
dsCsvReport.AR2sLogData[4][5]  :=DSHmiStationDisplayInfo[4].sStationSequenceRecipeDescription;(*Sequences Recipe*)
dsCsvReport.AR2sLogData[4][6]  :='N/A';(*Sub Recipe*)
dsCsvReport.AR2sLogData[4][7]  :=DSHmiStationDisplayInfo[4].sStationSubDescription;(*Sub Recipe*)
dsCsvReport.AR2sLogData[4][8]  :=INT_TO_STRING(ARDsStnMinMaxEffTimeDisplay[4].iMinTime);(*Minimum Time*)
dsCsvReport.AR2sLogData[4][9]  :='N/A';(*Minimum Time*)
dsCsvReport.AR2sLogData[4][10]  :=INT_TO_STRING(ARDsStnMinMaxEffTimeDisplay[4].iMaxTime);(*Maximum Time*)
dsCsvReport.AR2sLogData[4][11] :='N/A';(*Maximum Time*)
dsCsvReport.AR2sLogData[4][12] :=INT_TO_STRING(ARDsStnMinMaxEffTimeDisplay[4].iEffTime);(*Effective Time*)
dsCsvReport.AR2sLogData[4][13] :='N/A';(*Effective Time*)
dsCsvReport.AR2sLogData[4][14] :=REAL_TO_STRING(ARrStnTempSV[4]);(*Temperature SV*)
dsCsvReport.AR2sLogData[4][15] :=REAL_TO_STRING(ARrStnTempPV[4]);(*Temperature PV*)
dsCsvReport.AR2sLogData[4][16] :=INT_TO_STRING(ARDsStnSeqProcessCtrl[4].Out_DSStnSeqProOutput.i3ProTankBtmUsAPwrPercent);(*U/Sonic Bottom A Power SV*)
dsCsvReport.AR2sLogData[4][17]:=INT_TO_STRING(ARiUsPowerPV_percent[4]);(*U/Sonic Bottom A Power PV*)
dsCsvReport.AR2sLogData[4][18]:='N/A';(*U/Sonic Bottom A Frequency SV*)
dsCsvReport.AR2sLogData[4][19]:=INT_TO_STRING(iDisplayFreqUs[4]);(*U/Sonic Bottom A Frequency PV*)
dsCsvReport.AR2sLogData[4][20]:='N/A';(*U/Sonic Bottom B Power SV*)
dsCsvReport.AR2sLogData[4][21]:='N/A';(*U/Sonic Bottom B Power PV*)
dsCsvReport.AR2sLogData[4][22]:='N/A';(*U/Sonic Bottom B Frequency SV*)
dsCsvReport.AR2sLogData[4][23]:='N/A';(*U/Sonic Bottom B Frequency PV*)
dsCsvReport.AR2sLogData[4][24]:='N/A';(*U/Sonic Side A Power SV*)
dsCsvReport.AR2sLogData[4][25]:='N/A';(*U/Sonic Side A Power PV*)
dsCsvReport.AR2sLogData[4][26]:='N/A';(*U/Sonic Side A Frequency SV*)
dsCsvReport.AR2sLogData[4][27]:='N/A';(*U/Sonic Side A Frequency PV*)
dsCsvReport.AR2sLogData[4][28]:='N/A';(*U/Sonic Side B Power SV*)
dsCsvReport.AR2sLogData[4][29]:='N/A';(*U/Sonic Side B Power PV*)
dsCsvReport.AR2sLogData[4][30]:='N/A';(*U/Sonic Side B Frequency SV*)
dsCsvReport.AR2sLogData[4][31]:='N/A';(*U/Sonic Side B Frequency PV*)
dsCsvReport.AR2sLogData[4][32]:='N/A';(*Vacuum SV*)
dsCsvReport.AR2sLogData[4][33]:='N/A';(*Vacuum PV*)
dsCsvReport.AR2sLogData[4][34]:='N/A';(*Conductivity SV*)
dsCsvReport.AR2sLogData[4][35]:=REAL_TO_STRING(ARrStnConductivityPV[4]);(*Conductivity PV*)
dsCsvReport.AR2sLogData[4][36]:='N/A';(*Pump Flow SV*)
dsCsvReport.AR2sLogData[4][37]:=REAL_TO_STRING(ARrStnFilterPressurePV[4]);(*Pump Flow PV*)
dsCsvReport.AR2sLogData[4][38]:='N/A';(*Resistivity SV*)
dsCsvReport.AR2sLogData[4][39]:='N/A';(*Resistivity PV*)
dsCsvReport.AR2sLogData[4][40]:='N/A';(*PH SV*)
dsCsvReport.AR2sLogData[4][41]:='N/A'; (*PH PV*)
dsCsvReport.AR2sLogData[4][42]:='N/A';(*Quality*)
dsCsvReport.AR2sLogData[4][43]:=DSStnBasketInfo[4].sProductQuality;(*Quality*)
dsCsvReport.AR2sLogData[4][44]:=INT_TO_STRING(ARDsStnSeqProcessCtrl[4].Out_iCurrentProcessTime);(*Actual Time*)
dsCsvReport.AR2sLogData[4][45]:='N/A';(*Actual Time*)               

                         
// Data log info STN 05 ( NINE ROW )5 -US CLEANING
dsCsvReport.AR2sLogData[5][1]  :=sTime;
dsCsvReport.AR2sLogData[5][2]  :='N/A';(*Station*)
dsCsvReport.AR2sLogData[5][3]  :='5-SONIC CLEANING';(*Station*)
dsCsvReport.AR2sLogData[5][4]  :='N/A';(*Sequences Recipe*)
dsCsvReport.AR2sLogData[5][5]  :=DSHmiStationDisplayInfo[5].sStationSequenceRecipeDescription;(*Sequences Recipe*)
dsCsvReport.AR2sLogData[5][6]  :='N/A';(*Sub Recipe*)
dsCsvReport.AR2sLogData[5][7]  :=DSHmiStationDisplayInfo[5].sStationSubDescription;(*Sub Recipe*)
dsCsvReport.AR2sLogData[5][8]  :=INT_TO_STRING(ARDsStnMinMaxEffTimeDisplay[5].iMinTime);(*Minimum Time*)
dsCsvReport.AR2sLogData[5][9]  :='N/A';(*Minimum Time*)
dsCsvReport.AR2sLogData[5][10]  :=INT_TO_STRING(ARDsStnMinMaxEffTimeDisplay[5].iMaxTime);(*Maximum Time*)
dsCsvReport.AR2sLogData[5][11] :='N/A';(*Maximum Time*)
dsCsvReport.AR2sLogData[5][12] :=INT_TO_STRING(ARDsStnMinMaxEffTimeDisplay[5].iEffTime);(*Effective Time*)
dsCsvReport.AR2sLogData[5][13] :='N/A';(*Effective Time*)
dsCsvReport.AR2sLogData[5][14] :=REAL_TO_STRING(ARrStnTempSV[5]);(*Temperature SV*)
dsCsvReport.AR2sLogData[5][15] :=REAL_TO_STRING(ARrStnTempPV[5]);(*Temperature PV*)
dsCsvReport.AR2sLogData[5][16] :=INT_TO_STRING(ARDsStnSeqProcessCtrl[5].Out_DSStnSeqProOutput.i3ProTankBtmUsAPwrPercent);(*U/Sonic Bottom A Power SV*)
dsCsvReport.AR2sLogData[5][17]:=INT_TO_STRING(ARiUsPowerPV_percent[5]);(*U/Sonic Bottom A Power PV*)
dsCsvReport.AR2sLogData[5][18]:='N/A';(*U/Sonic Bottom A Frequency SV*)
dsCsvReport.AR2sLogData[5][19]:=INT_TO_STRING(iDisplayFreqUs[5]);(*U/Sonic Bottom A Frequency PV*)
dsCsvReport.AR2sLogData[5][20]:='N/A';(*U/Sonic Bottom B Power SV*)
dsCsvReport.AR2sLogData[5][21]:='N/A';(*U/Sonic Bottom B Power PV*)
dsCsvReport.AR2sLogData[5][22]:='N/A';(*U/Sonic Bottom B Frequency SV*)
dsCsvReport.AR2sLogData[5][23]:='N/A';(*U/Sonic Bottom B Frequency PV*)
dsCsvReport.AR2sLogData[5][24]:='N/A';(*U/Sonic Side A Power SV*)
dsCsvReport.AR2sLogData[5][25]:='N/A';(*U/Sonic Side A Power PV*)
dsCsvReport.AR2sLogData[5][26]:='N/A';(*U/Sonic Side A Frequency SV*)
dsCsvReport.AR2sLogData[5][27]:='N/A';(*U/Sonic Side A Frequency PV*)
dsCsvReport.AR2sLogData[5][28]:='N/A';(*U/Sonic Side B Power SV*)
dsCsvReport.AR2sLogData[5][29]:='N/A';(*U/Sonic Side B Power PV*)
dsCsvReport.AR2sLogData[5][30]:='N/A';(*U/Sonic Side B Frequency SV*)
dsCsvReport.AR2sLogData[5][31]:='N/A';(*U/Sonic Side B Frequency PV*)
dsCsvReport.AR2sLogData[5][32]:='N/A';(*Vacuum SV*)
dsCsvReport.AR2sLogData[5][33]:='N/A';(*Vacuum PV*)
dsCsvReport.AR2sLogData[5][34]:='N/A';(*Conductivity SV*)
dsCsvReport.AR2sLogData[5][35]:=REAL_TO_STRING(ARrStnConductivityPV[5]);(*Conductivity PV*)
dsCsvReport.AR2sLogData[5][36]:='N/A';(*Pump Flow SV*)
dsCsvReport.AR2sLogData[5][37]:=REAL_TO_STRING(ARrStnFilterPressurePV[5]);(*Pump Flow PV*)
dsCsvReport.AR2sLogData[5][38]:='N/A';(*Resistivity SV*)
dsCsvReport.AR2sLogData[5][39]:='N/A';(*Resistivity PV*)
dsCsvReport.AR2sLogData[5][40]:='N/A';(*PH SV*)
dsCsvReport.AR2sLogData[5][41]:='N/A'; (*PH PV*)
dsCsvReport.AR2sLogData[5][42]:='N/A';(*Quality*)
dsCsvReport.AR2sLogData[5][43]:=DSStnBasketInfo[5].sProductQuality;(*Quality*)
dsCsvReport.AR2sLogData[5][44]:=INT_TO_STRING(ARDsStnSeqProcessCtrl[5].Out_iCurrentProcessTime);(*Actual Time*)
dsCsvReport.AR2sLogData[5][45]:='N/A';(*Actual Time*)    
               
           

// Data log info STN 06 ( NINE ROW )6-RINSING
dsCsvReport.AR2sLogData[6][1]  :=sTime;
dsCsvReport.AR2sLogData[6][2]  :='N/A';(*Station*)
dsCsvReport.AR2sLogData[6][3]  :='6-RINSING';(*Station*)
dsCsvReport.AR2sLogData[6][4]  :='N/A';(*Sequences Recipe*)
dsCsvReport.AR2sLogData[6][5]  :=DSHmiStationDisplayInfo[6].sStationSequenceRecipeDescription;(*Sequences Recipe*)
dsCsvReport.AR2sLogData[6][6]  :='N/A';(*Sub Recipe*)
dsCsvReport.AR2sLogData[6][7]  :=DSHmiStationDisplayInfo[6].sStationSubDescription;(*Sub Recipe*)
dsCsvReport.AR2sLogData[6][8]  :=INT_TO_STRING(ARDsStnMinMaxEffTimeDisplay[6].iMinTime);(*Minimum Time*)
dsCsvReport.AR2sLogData[6][9]  :='N/A';(*Minimum Time*)
dsCsvReport.AR2sLogData[6][10]  :=INT_TO_STRING(ARDsStnMinMaxEffTimeDisplay[6].iMaxTime);(*Maximum Time*)
dsCsvReport.AR2sLogData[6][11] :='N/A';(*Maximum Time*)
dsCsvReport.AR2sLogData[6][12] :=INT_TO_STRING(ARDsStnMinMaxEffTimeDisplay[6].iEffTime);(*Effective Time*)
dsCsvReport.AR2sLogData[6][13] :='N/A';(*Effective Time*)
dsCsvReport.AR2sLogData[6][14] :=REAL_TO_STRING(ARrStnTempSV[6]);(*Temperature SV*)
dsCsvReport.AR2sLogData[6][15] :=REAL_TO_STRING(ARrStnTempPV[6]);(*Temperature PV*)
dsCsvReport.AR2sLogData[6][16] :=INT_TO_STRING(ARDsStnSeqProcessCtrl[6].Out_DSStnSeqProOutput.i3ProTankBtmUsAPwrPercent);(*U/Sonic Bottom A Power SV*)
dsCsvReport.AR2sLogData[6][17]:=INT_TO_STRING(ARiMegaPowerPV_percent[3]);(*U/Sonic Bottom A Power PV*)
dsCsvReport.AR2sLogData[6][18]:='N/A';(*U/Sonic Bottom A Frequency SV*)
dsCsvReport.AR2sLogData[6][19]:=INT_TO_STRING(DSV2ModbusControl2.wModbusData[9]);(*U/Sonic Bottom A Frequency PV*)
dsCsvReport.AR2sLogData[6][20]:='N/A';(*U/Sonic Bottom B Power SV*)
dsCsvReport.AR2sLogData[6][21]:='N/A';(*U/Sonic Bottom B Power PV*)
dsCsvReport.AR2sLogData[6][22]:='N/A';(*U/Sonic Bottom B Frequency SV*)
dsCsvReport.AR2sLogData[6][23]:='N/A';(*U/Sonic Bottom B Frequency PV*)
dsCsvReport.AR2sLogData[6][24]:='N/A';(*U/Sonic Side A Power SV*)
dsCsvReport.AR2sLogData[6][25]:='N/A';(*U/Sonic Side A Power PV*)
dsCsvReport.AR2sLogData[6][26]:='N/A';(*U/Sonic Side A Frequency SV*)
dsCsvReport.AR2sLogData[6][27]:='N/A';(*U/Sonic Side A Frequency PV*)
dsCsvReport.AR2sLogData[6][28]:='N/A';(*U/Sonic Side B Power SV*)
dsCsvReport.AR2sLogData[6][29]:='N/A';(*U/Sonic Side B Power PV*)
dsCsvReport.AR2sLogData[6][30]:='N/A';(*U/Sonic Side B Frequency SV*)
dsCsvReport.AR2sLogData[6][31]:='N/A';(*U/Sonic Side B Frequency PV*)
dsCsvReport.AR2sLogData[6][32]:='N/A';(*Vacuum SV*)
dsCsvReport.AR2sLogData[6][33]:='N/A';(*Vacuum PV*)
dsCsvReport.AR2sLogData[6][34]:='N/A';(*Conductivity SV*)
dsCsvReport.AR2sLogData[6][35]:=REAL_TO_STRING(ARrStnConductivityPV[6]);(*Conductivity PV*)
dsCsvReport.AR2sLogData[6][36]:='N/A';(*Pump Flow SV*)
dsCsvReport.AR2sLogData[6][37]:=REAL_TO_STRING(ARrStnFilterPressurePV[6]);(*Pump Flow PV*)
dsCsvReport.AR2sLogData[6][38]:='N/A';(*Resistivity SV*)
dsCsvReport.AR2sLogData[6][39]:='N/A';(*Resistivity PV*)
dsCsvReport.AR2sLogData[6][40]:='N/A';(*PH SV*)
dsCsvReport.AR2sLogData[6][41]:='N/A'; (*PH PV*)
dsCsvReport.AR2sLogData[6][42]:='N/A';(*Quality*)
dsCsvReport.AR2sLogData[6][43]:=DSStnBasketInfo[6].sProductQuality;(*Quality*)
dsCsvReport.AR2sLogData[6][44]:=INT_TO_STRING(ARDsStnSeqProcessCtrl[6].Out_iCurrentProcessTime);(*Actual Time*)
dsCsvReport.AR2sLogData[6][45]:='N/A';(*Actual Time*)                      


// Data log info STN 07 ( NINE ROW )7- FINE RINSING
dsCsvReport.AR2sLogData[7][1]  :=sTime;(*Station*)
dsCsvReport.AR2sLogData[7][2]  :='N/A';(*Station*)
dsCsvReport.AR2sLogData[7][3]  :='7-FINE RINSING';(*Station*)
dsCsvReport.AR2sLogData[7][4]  :='N/A';(*Sequences Recipe*)
dsCsvReport.AR2sLogData[7][5]  :=DSHmiStationDisplayInfo[7].sStationSequenceRecipeDescription;(*Sequences Recipe*)
dsCsvReport.AR2sLogData[7][6]  :='N/A';(*Sub Recipe*)
dsCsvReport.AR2sLogData[7][7]  :=DSHmiStationDisplayInfo[7].sStationSubDescription;(*Sub Recipe*)
dsCsvReport.AR2sLogData[7][8]  :=INT_TO_STRING(ARDsStnMinMaxEffTimeDisplay[7].iMinTime);(*Minimum Time*)
dsCsvReport.AR2sLogData[7][9]  :='N/A';(*Minimum Time*)
dsCsvReport.AR2sLogData[7][10]  :=INT_TO_STRING(ARDsStnMinMaxEffTimeDisplay[7].iMaxTime);(*Maximum Time*)
dsCsvReport.AR2sLogData[7][11] :='N/A';(*Maximum Time*)
dsCsvReport.AR2sLogData[7][12] :=INT_TO_STRING(ARDsStnMinMaxEffTimeDisplay[7].iEffTime);(*Effective Time*)
dsCsvReport.AR2sLogData[7][13] :='N/A';(*Effective Time*)
dsCsvReport.AR2sLogData[7][14] :=REAL_TO_STRING(ARrStnTempSV[7]);(*Temperature SV*)
dsCsvReport.AR2sLogData[7][15] :=REAL_TO_STRING(ARrStnTempPV[7]);(*Temperature PV*)
dsCsvReport.AR2sLogData[7][16] :=INT_TO_STRING(ARDsStnSeqProcessCtrl[7].Out_DSStnSeqProOutput.i3ProTankBtmUsAPwrPercent);(*U/Sonic Bottom A Power SV*)
dsCsvReport.AR2sLogData[7][17]:=INT_TO_STRING(ARiUsPowerPV_percent[7]);(*U/Sonic Bottom A Power PV*)
dsCsvReport.AR2sLogData[7][18]:='N/A';(*U/Sonic Bottom A Frequency SV*)
dsCsvReport.AR2sLogData[7][19]:=INT_TO_STRING(iDisplayFreqUs[7]);(*U/Sonic Bottom A Frequency PV*)
dsCsvReport.AR2sLogData[7][20]:='N/A';(*U/Sonic Bottom B Power SV*)
dsCsvReport.AR2sLogData[7][21]:='N/A';(*U/Sonic Bottom B Power PV*)
dsCsvReport.AR2sLogData[7][22]:='N/A';(*U/Sonic Bottom B Frequency SV*)
dsCsvReport.AR2sLogData[7][23]:='N/A';(*U/Sonic Bottom B Frequency PV*)
dsCsvReport.AR2sLogData[7][24]:='N/A';(*U/Sonic Side A Power SV*)
dsCsvReport.AR2sLogData[7][25]:='N/A';(*U/Sonic Side A Power PV*)
dsCsvReport.AR2sLogData[7][26]:='N/A';(*U/Sonic Side A Frequency SV*)
dsCsvReport.AR2sLogData[7][27]:='N/A';(*U/Sonic Side A Frequency PV*)
dsCsvReport.AR2sLogData[7][28]:='N/A';(*U/Sonic Side B Power SV*)
dsCsvReport.AR2sLogData[7][29]:='N/A';(*U/Sonic Side B Power PV*)
dsCsvReport.AR2sLogData[7][30]:='N/A';(*U/Sonic Side B Frequency SV*)
dsCsvReport.AR2sLogData[7][31]:='N/A';(*U/Sonic Side B Frequency PV*)
dsCsvReport.AR2sLogData[7][32]:='N/A';(*Vacuum SV*)
dsCsvReport.AR2sLogData[7][33]:='N/A';(*Vacuum PV*)
dsCsvReport.AR2sLogData[7][34]:='N/A';(*Conductivity SV*)
dsCsvReport.AR2sLogData[7][35]:=REAL_TO_STRING(ARrStnConductivityPV[7]);(*Conductivity PV*)
dsCsvReport.AR2sLogData[7][36]:='N/A';(*Pump Flow SV*)
dsCsvReport.AR2sLogData[7][37]:=REAL_TO_STRING(ARrStnFilterPressurePV[7]);(*Pump Flow PV*)
dsCsvReport.AR2sLogData[7][38]:='N/A';(*Resistivity SV*)
dsCsvReport.AR2sLogData[7][39]:='N/A';(*Resistivity PV*)
dsCsvReport.AR2sLogData[7][40]:='N/A';(*PH SV*)
dsCsvReport.AR2sLogData[7][41]:='N/A'; (*PH PV*)
dsCsvReport.AR2sLogData[7][42]:='N/A';(*Quality*)
dsCsvReport.AR2sLogData[7][43]:=DSStnBasketInfo[7].sProductQuality;(*Quality*)
dsCsvReport.AR2sLogData[7][44]:=INT_TO_STRING(ARDsStnSeqProcessCtrl[7].Out_iCurrentProcessTime);(*Actual Time*)
dsCsvReport.AR2sLogData[7][45]:='N/A';(*Actual Time*) 
                             

// Data log info STN 08 ( NINE ROW )8- FINE RINSING
dsCsvReport.AR2sLogData[8][1]  :=sTime;(*Station*)
dsCsvReport.AR2sLogData[8][2]  :='N/A';(*Station*)
dsCsvReport.AR2sLogData[8][3]  :='8-FINE RINSING';(*Station*)
dsCsvReport.AR2sLogData[8][4]  :='N/A';(*Sequences Recipe*)
dsCsvReport.AR2sLogData[8][5]  :=DSHmiStationDisplayInfo[8].sStationSequenceRecipeDescription;(*Sequences Recipe*)
dsCsvReport.AR2sLogData[8][6]  :='N/A';(*Sub Recipe*)
dsCsvReport.AR2sLogData[8][7]  :=DSHmiStationDisplayInfo[8].sStationSubDescription;(*Sub Recipe*)
dsCsvReport.AR2sLogData[8][8]  :=INT_TO_STRING(ARDsStnMinMaxEffTimeDisplay[8].iMinTime);(*Minimum Time*)
dsCsvReport.AR2sLogData[8][9]  :='N/A';(*Minimum Time*)
dsCsvReport.AR2sLogData[8][10]  :=INT_TO_STRING(ARDsStnMinMaxEffTimeDisplay[8].iMaxTime);(*Maximum Time*)
dsCsvReport.AR2sLogData[8][11] :='N/A';(*Maximum Time*)
dsCsvReport.AR2sLogData[8][12] :=INT_TO_STRING(ARDsStnMinMaxEffTimeDisplay[8].iEffTime);(*Effective Time*)
dsCsvReport.AR2sLogData[8][13] :='N/A';(*Effective Time*)
dsCsvReport.AR2sLogData[8][14] :=REAL_TO_STRING(ARrStnTempSV[8]);(*Temperature SV*)
dsCsvReport.AR2sLogData[8][15] :=REAL_TO_STRING(ARrStnTempPV[8]);(*Temperature PV*)
dsCsvReport.AR2sLogData[8][16] :=INT_TO_STRING(ARDsStnSeqProcessCtrl[8].Out_DSStnSeqProOutput.i3ProTankBtmUsAPwrPercent);(*U/Sonic Bottom A Power SV*)
dsCsvReport.AR2sLogData[8][17]:=INT_TO_STRING(ARiUsPowerPV_percent[8]);(*U/Sonic Bottom A Power PV*)
dsCsvReport.AR2sLogData[8][18]:='N/A';(*U/Sonic Bottom A Frequency SV*)
dsCsvReport.AR2sLogData[8][19]:=INT_TO_STRING(iDisplayFreqUs[8]);(*U/Sonic Bottom A Frequency PV*)
dsCsvReport.AR2sLogData[8][20]:='N/A';(*U/Sonic Bottom B Power SV*)
dsCsvReport.AR2sLogData[8][21]:='N/A';(*U/Sonic Bottom B Power PV*)
dsCsvReport.AR2sLogData[8][22]:='N/A';(*U/Sonic Bottom B Frequency SV*)
dsCsvReport.AR2sLogData[8][23]:='N/A';(*U/Sonic Bottom B Frequency PV*)
dsCsvReport.AR2sLogData[8][24]:='N/A';(*U/Sonic Side A Power SV*)
dsCsvReport.AR2sLogData[8][25]:='N/A';(*U/Sonic Side A Power PV*)
dsCsvReport.AR2sLogData[8][26]:='N/A';(*U/Sonic Side A Frequency SV*)
dsCsvReport.AR2sLogData[8][27]:='N/A';(*U/Sonic Side A Frequency PV*)
dsCsvReport.AR2sLogData[8][28]:='N/A';(*U/Sonic Side B Power SV*)
dsCsvReport.AR2sLogData[8][29]:='N/A';(*U/Sonic Side B Power PV*)
dsCsvReport.AR2sLogData[8][30]:='N/A';(*U/Sonic Side B Frequency SV*)
dsCsvReport.AR2sLogData[8][31]:='N/A';(*U/Sonic Side B Frequency PV*)
dsCsvReport.AR2sLogData[8][32]:='N/A';(*Vacuum SV*)
dsCsvReport.AR2sLogData[8][33]:='N/A';(*Vacuum PV*)
dsCsvReport.AR2sLogData[8][34]:='N/A';(*Conductivity SV*)
dsCsvReport.AR2sLogData[8][35]:=REAL_TO_STRING(ARrStnConductivityPV[8]);(*Conductivity PV*)
dsCsvReport.AR2sLogData[8][36]:='N/A';(*Pump Flow SV*)
dsCsvReport.AR2sLogData[8][37]:=REAL_TO_STRING(ARrStnFilterPressurePV[8]);(*Pump Flow PV*)
dsCsvReport.AR2sLogData[8][38]:='N/A';(*Resistivity SV*)
dsCsvReport.AR2sLogData[8][39]:='N/A';(*Resistivity PV*)
dsCsvReport.AR2sLogData[8][40]:='N/A';(*PH SV*)
dsCsvReport.AR2sLogData[8][41]:='N/A'; (*PH PV*)
dsCsvReport.AR2sLogData[8][42]:='N/A';(*Quality*)
dsCsvReport.AR2sLogData[8][43]:=DSStnBasketInfo[8].sProductQuality;(*Quality*)
dsCsvReport.AR2sLogData[8][44]:=INT_TO_STRING(ARDsStnSeqProcessCtrl[8].Out_iCurrentProcessTime);(*Actual Time*)
dsCsvReport.AR2sLogData[8][45]:='N/A';(*Actual Time*)                        

// Data log info STN 09 ( NINE ROW )9-INFRARED DRYER
dsCsvReport.AR2sLogData[9][1]  :=sTime;(*Station*)
dsCsvReport.AR2sLogData[9][2]  :='N/A';(*Station*)
dsCsvReport.AR2sLogData[9][3]  :='9-PRECISION RINSING';(*Station*)
dsCsvReport.AR2sLogData[9][4]  :='N/A';(*Sequences Recipe*)
dsCsvReport.AR2sLogData[9][5]  :=DSHmiStationDisplayInfo[9].sStationSequenceRecipeDescription;(*Sequences Recipe*)
dsCsvReport.AR2sLogData[9][6]  :='N/A';(*Sub Recipe*)
dsCsvReport.AR2sLogData[9][7]  :=DSHmiStationDisplayInfo[9].sStationSubDescription;(*Sub Recipe*)
dsCsvReport.AR2sLogData[9][8]  :=INT_TO_STRING(ARDsStnMinMaxEffTimeDisplay[9].iMinTime);(*Minimum Time*)
dsCsvReport.AR2sLogData[9][9]  :='N/A';(*Minimum Time*)
dsCsvReport.AR2sLogData[9][10] :=INT_TO_STRING(ARDsStnMinMaxEffTimeDisplay[9].iMaxTime);(*Maximum Time*)
dsCsvReport.AR2sLogData[9][11] :='N/A';(*Maximum Time*)
dsCsvReport.AR2sLogData[9][12] :=INT_TO_STRING(ARDsStnMinMaxEffTimeDisplay[9].iEffTime);(*Effective Time*)
dsCsvReport.AR2sLogData[9][13] :='N/A';(*Effective Time*)
dsCsvReport.AR2sLogData[9][14] :=REAL_TO_STRING(ARrStnTempSV[9]);(*Temperature SV*)
dsCsvReport.AR2sLogData[9][15] :=REAL_TO_STRING(ARrStnTempPV[9]);(*Temperature PV*)
dsCsvReport.AR2sLogData[9][16] :='';(*U/Sonic Bottom A Power SV*)
dsCsvReport.AR2sLogData[9][17]:='';(*U/Sonic Bottom A Power PV*)
dsCsvReport.AR2sLogData[9][18]:='N/A';(*U/Sonic Bottom A Frequency SV*)
dsCsvReport.AR2sLogData[9][19]:='';(*U/Sonic Bottom A Frequency PV*)
dsCsvReport.AR2sLogData[9][20]:='N/A';(*U/Sonic Bottom B Power SV*)
dsCsvReport.AR2sLogData[9][21]:='N/A';(*U/Sonic Bottom B Power PV*)
dsCsvReport.AR2sLogData[9][22]:='N/A';(*U/Sonic Bottom B Frequency SV*)
dsCsvReport.AR2sLogData[9][23]:='N/A';(*U/Sonic Bottom B Frequency PV*)
dsCsvReport.AR2sLogData[9][24]:='N/A';(*U/Sonic Side A Power SV*)
dsCsvReport.AR2sLogData[9][25]:='N/A';(*U/Sonic Side A Power PV*)
dsCsvReport.AR2sLogData[9][26]:='N/A';(*U/Sonic Side A Frequency SV*)
dsCsvReport.AR2sLogData[9][27]:='N/A';(*U/Sonic Side A Frequency PV*)
dsCsvReport.AR2sLogData[9][28]:='N/A';(*U/Sonic Side B Power SV*)
dsCsvReport.AR2sLogData[9][29]:='N/A';(*U/Sonic Side B Power PV*)
dsCsvReport.AR2sLogData[9][30]:='N/A';(*U/Sonic Side B Frequency SV*)
dsCsvReport.AR2sLogData[9][31]:='N/A';(*U/Sonic Side B Frequency PV*)
dsCsvReport.AR2sLogData[9][32]:='N/A';(*Vacuum SV*)
dsCsvReport.AR2sLogData[9][33]:='N/A';(*Vacuum PV*)
dsCsvReport.AR2sLogData[9][34]:='N/A';(*Conductivity SV*)
dsCsvReport.AR2sLogData[9][35]:=REAL_TO_STRING(ARrStnConductivityPV[9]);(*Conductivity PV*)
dsCsvReport.AR2sLogData[9][36]:='N/A';(*Pump Flow SV*)
dsCsvReport.AR2sLogData[9][37]:=REAL_TO_STRING(ARrStnFilterPressurePV[9]);(*Pump Flow PV*)
dsCsvReport.AR2sLogData[9][38]:='N/A';(*Resistivity SV*)
dsCsvReport.AR2sLogData[9][39]:='N/A';(*Resistivity PV*)
dsCsvReport.AR2sLogData[9][40]:='N/A';(*PH SV*)
dsCsvReport.AR2sLogData[9][41]:='N/A'; (*PH PV*)
dsCsvReport.AR2sLogData[9][42]:='N/A';(*Quality*)
dsCsvReport.AR2sLogData[9][43]:=DSStnBasketInfo[9].sProductQuality;(*Quality*)
dsCsvReport.AR2sLogData[9][44]:=INT_TO_STRING(ARDsStnSeqProcessCtrl[9].Out_iCurrentProcessTime);(*Actual Time*)
dsCsvReport.AR2sLogData[9][45]:='N/A';(*Actual Time*)                        
                  

// Data LOG info STN 10 ( NINE ROW )
dsCsvReport.AR2sLogData[10][1]  :=sTime;(*Station*)
dsCsvReport.AR2sLogData[10][2]  :='N/A';(*Station*)
dsCsvReport.AR2sLogData[10][3]  :='10-INFRARED DRYER';(*Station*)
dsCsvReport.AR2sLogData[10][4]  :='N/A';(*Sequences Recipe*)
dsCsvReport.AR2sLogData[10][5]  :=DSHmiStationDisplayInfo[10].sStationSequenceRecipeDescription;(*Sequences Recipe*)
dsCsvReport.AR2sLogData[10][6]  :='N/A';(*Sub Recipe*)
dsCsvReport.AR2sLogData[10][7]  :=DSHmiStationDisplayInfo[10].sStationSubDescription;(*Sub Recipe*)
dsCsvReport.AR2sLogData[10][8]  :=INT_TO_STRING(ARDsStnMinMaxEffTimeDisplay[10].iMinTime);(*Minimum Time*)
dsCsvReport.AR2sLogData[10][9]  :='N/A';(*Minimum Time*)
dsCsvReport.AR2sLogData[10][10]  :=INT_TO_STRING(ARDsStnMinMaxEffTimeDisplay[10].iMaxTime);(*Maximum Time*)
dsCsvReport.AR2sLogData[10][11] :='N/A';(*Maximum Time*)
dsCsvReport.AR2sLogData[10][12] :=INT_TO_STRING(ARDsStnMinMaxEffTimeDisplay[10].iEffTime);(*Effective Time*)
dsCsvReport.AR2sLogData[10][13] :='N/A';(*Effective Time*)
dsCsvReport.AR2sLogData[10][14] :=REAL_TO_STRING(ARrStnTempSV[10]);(*Temperature SV*)
dsCsvReport.AR2sLogData[10][15] :=REAL_TO_STRING(ARrStnTempPV[10]);(*Temperature PV*)
dsCsvReport.AR2sLogData[10][16] :='';(*U/Sonic Bottom A Power SV*)
dsCsvReport.AR2sLogData[10][17]:='';(*U/Sonic Bottom A Power PV*)
dsCsvReport.AR2sLogData[10][18]:='N/A';(*U/Sonic Bottom A Frequency SV*)
dsCsvReport.AR2sLogData[10][19]:='';(*U/Sonic Bottom A Frequency PV*)
dsCsvReport.AR2sLogData[10][20]:='N/A';(*U/Sonic Bottom B Power SV*)
dsCsvReport.AR2sLogData[10][21]:='N/A';(*U/Sonic Bottom B Power PV*)
dsCsvReport.AR2sLogData[10][22]:='N/A';(*U/Sonic Bottom B Frequency SV*)
dsCsvReport.AR2sLogData[10][23]:='N/A';(*U/Sonic Bottom B Frequency PV*)
dsCsvReport.AR2sLogData[10][24]:='N/A';(*U/Sonic Side A Power SV*)
dsCsvReport.AR2sLogData[10][25]:='N/A';(*U/Sonic Side A Power PV*)
dsCsvReport.AR2sLogData[10][26]:='N/A';(*U/Sonic Side A Frequency SV*)
dsCsvReport.AR2sLogData[10][27]:='N/A';(*U/Sonic Side A Frequency PV*)
dsCsvReport.AR2sLogData[10][28]:='N/A';(*U/Sonic Side B Power SV*)
dsCsvReport.AR2sLogData[10][29]:='N/A';(*U/Sonic Side B Power PV*)
dsCsvReport.AR2sLogData[10][30]:='N/A';(*U/Sonic Side B Frequency SV*)
dsCsvReport.AR2sLogData[10][31]:='N/A';(*U/Sonic Side B Frequency PV*)
dsCsvReport.AR2sLogData[10][32]:='N/A';(*Vacuum SV*)
dsCsvReport.AR2sLogData[10][33]:='N/A';(*Vacuum PV*)
dsCsvReport.AR2sLogData[10][34]:='N/A';(*Conductivity SV*)
dsCsvReport.AR2sLogData[10][35]:='N/A';(*Conductivity PV*)
dsCsvReport.AR2sLogData[10][36]:='N/A';(*Pump Flow SV*)
dsCsvReport.AR2sLogData[10][37]:='N/A';(*Pump Flow PV*)
dsCsvReport.AR2sLogData[10][38]:='N/A';(*Resistivity SV*)
dsCsvReport.AR2sLogData[10][39]:='N/A';(*Resistivity PV*)
dsCsvReport.AR2sLogData[10][40]:='N/A';(*PH SV*)
dsCsvReport.AR2sLogData[10][41]:='N/A'; (*PH PV*)
dsCsvReport.AR2sLogData[10][42]:='N/A';(*Quality*)
dsCsvReport.AR2sLogData[10][43]:=DSStnBasketInfo[10].sProductQuality;(*Quality*)
dsCsvReport.AR2sLogData[10][44]:=INT_TO_STRING(ARDsStnSeqProcessCtrl[10].Out_iCurrentProcessTime);(*Actual Time*)
dsCsvReport.AR2sLogData[10][45]:='N/A';(*Actual Time*)            




	sCsvFilePath								:= 'C:\JKS\report_csv\';
	udiCsvMRBCount								;	// The number of data set stored in MRB (MemoryRingBuffer)
	udiCsvMRBUsagePercent 						;	// Current Usage % in MRB (MemoryRingBuffer)

	// Check if thats a problem
	ARdsCsvErrorLog[1].sPathAndFilename;
	ARdsCsvErrorLog[1].eLogAction;
	ARdsCsvErrorLog[1].sLogString;
	ARdsCsvErrorLog[1].iCaseid;
	ARdsCsvErrorLog[1].udiErrorId;

	ARdsCsvErrorLog[2].sPathAndFilename;
	ARdsCsvErrorLog[2].eLogAction;
	ARdsCsvErrorLog[2].sLogString;
	ARdsCsvErrorLog[2].iCaseid;
	ARdsCsvErrorLog[2].udiErrorId;

END_PROGRAM

// ---- POUs/MainProgram/DataManagement_Barcode/Log_BasketTimeInOut.TcPOU
PROGRAM Log_BasketTimeInOut
VAR
	ARbLdBasketAvailibilityRE	: ARRAY [0..iLdStnQty] OF R_TRIG;
	ARbUldBasketAvailibilityRE	: ARRAY [0..iUldStnQty] OF R_TRIG;
	ARbStnBasketAvailibilityRE	: ARRAY [0..iStnQty] OF R_TRIG;

	ARbLdBasketAvailibilityFE	: ARRAY [0..iLdStnQty] OF F_TRIG;
	ARbUldBasketAvailibilityFE	: ARRAY [0..iUldStnQty] OF F_TRIG;
	ARbStnBasketAvailibilityFE	: ARRAY [0..iStnQty] OF F_TRIG;

	ARtStnNotBasketAvailibility	: ARRAY [0..iStnQty] OF TON;
	ARtLdNotBasketAvailibility	: ARRAY [0..iLdStnQty] OF TON;
	ARtUldNotBasketAvailibility	: ARRAY [0..iUldStnQty] OF TON;

	ARbLdBasketInActivate		: ARRAY [0..iLdStnQty] OF BOOL;

	ARbStnBasketInActivate		: ARRAY [0..iStnQty] OF BOOL;
	ARbStnBasketOutActivate		: ARRAY [0..iStnQty] OF BOOL;
	ARbUldBasketInActivate		: ARRAY [0..iUldStnQty] OF BOOL;
	
END_VAR

ARbLdBasketAvailibilityRE[1](CLK:= AR2sDSCv_LdConfirmBasketInfo[1,4].bAvailibility, Q=> );			ARbLdBasketAvailibilityFE[1](CLK:= AR2sDSCv_LdConfirmBasketInfo[1,4].bAvailibility, Q=> );
ARbUldBasketAvailibilityRE[1](CLK:= AR2sDSCv_UldConfirmBasketInfo[1,1].bAvailibility, Q=> );		ARbUldBasketAvailibilityFE[1](CLK:= AR2sDSCv_UldConfirmBasketInfo[1,1].bAvailibility, Q=> );
//ARbUldBasketAvailibilityRE[2](CLK:= AR2sDSCv_UldConfirmBasketInfo[2,1].bAvailibility, Q=> );		ARbUldBasketAvailibilityFE[2](CLK:= AR2sDSCv_UldConfirmBasketInfo[2,1].bAvailibility, Q=> );

ARbStnBasketAvailibilityRE[1](CLK:= DSStnBasketInfo[1].bAvailibility, Q=> );				ARbStnBasketAvailibilityFE[1](CLK:= DSStnBasketInfo[1].bAvailibility, Q=> );
ARbStnBasketAvailibilityRE[2](CLK:= DSStnBasketInfo[2].bAvailibility, Q=> );				ARbStnBasketAvailibilityFE[2](CLK:= DSStnBasketInfo[2].bAvailibility, Q=> );
ARbStnBasketAvailibilityRE[3](CLK:= DSStnBasketInfo[3].bAvailibility, Q=> );				ARbStnBasketAvailibilityFE[3](CLK:= DSStnBasketInfo[3].bAvailibility, Q=> );
ARbStnBasketAvailibilityRE[4](CLK:= DSStnBasketInfo[4].bAvailibility, Q=> );				ARbStnBasketAvailibilityFE[4](CLK:= DSStnBasketInfo[4].bAvailibility, Q=> );
ARbStnBasketAvailibilityRE[5](CLK:= DSStnBasketInfo[5].bAvailibility, Q=> );				ARbStnBasketAvailibilityFE[5](CLK:= DSStnBasketInfo[5].bAvailibility, Q=> );
ARbStnBasketAvailibilityRE[6](CLK:= DSStnBasketInfo[6].bAvailibility, Q=> );				ARbStnBasketAvailibilityFE[6](CLK:= DSStnBasketInfo[6].bAvailibility, Q=> );
ARbStnBasketAvailibilityRE[7](CLK:= DSStnBasketInfo[7].bAvailibility, Q=> );				ARbStnBasketAvailibilityFE[7](CLK:= DSStnBasketInfo[7].bAvailibility, Q=> );
ARbStnBasketAvailibilityRE[8](CLK:= DSStnBasketInfo[8].bAvailibility, Q=> );				ARbStnBasketAvailibilityFE[8](CLK:= DSStnBasketInfo[8].bAvailibility, Q=> );
ARbStnBasketAvailibilityRE[9](CLK:= DSStnBasketInfo[9].bAvailibility, Q=> );				ARbStnBasketAvailibilityFE[9](CLK:= DSStnBasketInfo[9].bAvailibility, Q=> );
ARbStnBasketAvailibilityRE[10](CLK:= DSStnBasketInfo[10].bAvailibility, Q=> );				ARbStnBasketAvailibilityFE[10](CLK:= DSStnBasketInfo[10].bAvailibility, Q=> );
//ARbStnBasketAvailibilityRE[11](CLK:= DSStnBasketInfo[11].bAvailibility, Q=> );				ARbStnBasketAvailibilityFE[11](CLK:= DSStnBasketInfo[11].bAvailibility, Q=> );
//ARbStnBasketAvailibilityRE[12](CLK:= DSStnBasketInfo[12].bAvailibility, Q=> );				ARbStnBasketAvailibilityFE[12](CLK:= DSStnBasketInfo[12].bAvailibility, Q=> );

ARtLdNotBasketAvailibility[1](IN:=bAutoStartPb AND NOT AR2sDSCv_LdConfirmBasketInfo[1,4].bAvailibility , PT:=T#10S , Q=> , ET=> );

ARtUldNotBasketAvailibility[1](IN:=bAutoStartPb AND NOT AR2sDSCv_UldConfirmBasketInfo[1,1].bAvailibility , PT:=T#10s , Q=> , ET=> );
//ARtUldNotBasketAvailibility[2](IN:=bAutoStartPb AND NOT AR2sDSCv_UldConfirmBasketInfo[2,1].bAvailibility , PT:=T#10s , Q=> , ET=> );

ARtStnNotBasketAvailibility[1](IN:=bAutoStartPb AND NOT DSStnBasketInfo[1].bAvailibility , PT:=T#10s , Q=> , ET=> );
ARtStnNotBasketAvailibility[2](IN:=bAutoStartPb AND NOT DSStnBasketInfo[2].bAvailibility , PT:=T#10s , Q=> , ET=> );
ARtStnNotBasketAvailibility[3](IN:=bAutoStartPb AND NOT DSStnBasketInfo[3].bAvailibility , PT:=T#10s , Q=> , ET=> );
ARtStnNotBasketAvailibility[4](IN:=bAutoStartPb AND NOT DSStnBasketInfo[4].bAvailibility , PT:=T#10s , Q=> , ET=> );
ARtStnNotBasketAvailibility[5](IN:=bAutoStartPb AND NOT DSStnBasketInfo[5].bAvailibility , PT:=T#10s , Q=> , ET=> );
ARtStnNotBasketAvailibility[6](IN:=bAutoStartPb AND NOT DSStnBasketInfo[6].bAvailibility , PT:=T#10s , Q=> , ET=> );
ARtStnNotBasketAvailibility[7](IN:=bAutoStartPb AND NOT DSStnBasketInfo[7].bAvailibility , PT:=T#10s , Q=> , ET=> );
ARtStnNotBasketAvailibility[8](IN:=bAutoStartPb AND NOT DSStnBasketInfo[8].bAvailibility , PT:=T#10s , Q=> , ET=> );
ARtStnNotBasketAvailibility[9](IN:=bAutoStartPb AND NOT DSStnBasketInfo[9].bAvailibility , PT:=T#10s , Q=> , ET=> );
ARtStnNotBasketAvailibility[10](IN:=bAutoStartPb AND NOT DSStnBasketInfo[10].bAvailibility , PT:=T#10S , Q=> , ET=> );
//ARtStnNotBasketAvailibility[11](IN:=bAutoStartPb AND NOT DSStnBasketInfo[11].bAvailibility , PT:=T#10s , Q=> , ET=> );
//ARtStnNotBasketAvailibility[12](IN:=bAutoStartPb AND NOT DSStnBasketInfo[12].bAvailibility , PT:=T#10s , Q=> , ET=> );


IF (bAutoStartPb AND ARbLdBasketAvailibilityRE[1].Q )	THEN ARbLdBasketInActivate[1] 	:= TRUE; ARsLdBasketInTime[1] := DSLocalSystemTimeML.sCurrentDateTime;
ARiLdBasketProductRecipeBuffer[1] 	:= AR2sDSCv_LdConfirmBasketInfo[1,4].iProductRecipeNo; ARsLdBasketNoBuffer[1] 	:= AR2sDSCv_LdConfirmBasketInfo[1,4].sReservedInt; END_IF


IF bAutoStartPb AND ARbUldBasketAvailibilityRE[1].Q 	THEN ARbUldBasketInActivate[1] 	:= TRUE;  ARsUldBasketInTime[1] := DSLocalSystemTimeML.sCurrentDateTime;
ARiUldBasketProductRecipeBuffer[1] 	:= AR2sDSCv_UldConfirmBasketInfo[1,1].iProductRecipeNo; ARsUldBasketNoBuffer[1] 	:= AR2sDSCv_UldConfirmBasketInfo[1,1].sReservedInt; END_IF

//IF bAutoStartPb AND ARbUldBasketAvailibilityRE[2].Q 	THEN ARbUldBasketInActivate[2] 	:= TRUE; ARsUldBasketInTime[2] := DSLocalSystemTimeML.sCurrentDateTime;
//ARiUldBasketProductRecipeBuffer[2] 	:= AR2sDSCv_UldConfirmBasketInfo[2,1].iProductRecipeNo; ARsUldBasketNoBuffer[2] 	:= AR2sDSCv_UldConfirmBasketInfo[2,1].sReservedInt; END_IF


IF bAutoStartPb AND ARbStnBasketAvailibilityRE[1].Q 	THEN ARbStnBasketInActivate[1] 	:= TRUE; ARsStnBasketInTime[1] := DSLocalSystemTimeML.sCurrentDateTime;
ARiStnBasketProductRecipeBuffer[1] 	:= DSStnBasketInfo[1].iProductRecipeNo; ARsStnBasketNoBuffer[1] 	:= DSStnBasketInfo[1].sReservedInt; 	END_IF

IF bAutoStartPb AND ARbStnBasketAvailibilityFE[1].Q 	THEN ARbStnBasketOutActivate[1] 	:= TRUE; ARsStnBasketOutTime[1] := DSLocalSystemTimeML.sCurrentDateTime; 	END_IF

IF bAutoStartPb AND ARbStnBasketAvailibilityRE[2].Q 	THEN ARbStnBasketInActivate[2] 	:= TRUE; ARsStnBasketInTime[2] := DSLocalSystemTimeML.sCurrentDateTime;
ARiStnBasketProductRecipeBuffer[2] 	:= DSStnBasketInfo[2].iProductRecipeNo; ARsStnBasketNoBuffer[2] 	:= DSStnBasketInfo[2].sReservedInt; 	END_IF

IF bAutoStartPb AND ARbStnBasketAvailibilityFE[2].Q 	THEN ARbStnBasketOutActivate[2] 	:= TRUE; ARsStnBasketOutTime[2] := DSLocalSystemTimeML.sCurrentDateTime;	END_IF

IF bAutoStartPb AND ARbStnBasketAvailibilityRE[3].Q 	THEN ARbStnBasketInActivate[3] 	:= TRUE; ARsStnBasketInTime[3] := DSLocalSystemTimeML.sCurrentDateTime;;
ARiStnBasketProductRecipeBuffer[3] 	:= DSStnBasketInfo[3].iProductRecipeNo; ARsStnBasketNoBuffer[3] 	:= DSStnBasketInfo[3].sReservedInt; 	END_IF

IF bAutoStartPb AND ARbStnBasketAvailibilityFE[3].Q 	THEN ARbStnBasketOutActivate[3] 	:= TRUE; ARsStnBasketOutTime[3] := DSLocalSystemTimeML.sCurrentDateTime; 	END_IF

IF bAutoStartPb AND ARbStnBasketAvailibilityRE[4].Q 	THEN ARbStnBasketInActivate[4] 	:= TRUE; ARsStnBasketInTime[4] := DSLocalSystemTimeML.sCurrentDateTime;;
ARiStnBasketProductRecipeBuffer[4] 	:= DSStnBasketInfo[4].iProductRecipeNo; ARsStnBasketNoBuffer[4] 	:= DSStnBasketInfo[4].sReservedInt; 	END_IF

IF bAutoStartPb AND ARbStnBasketAvailibilityFE[4].Q 	THEN ARbStnBasketOutActivate[4] 	:= TRUE; ARsStnBasketOutTime[4] := DSLocalSystemTimeML.sCurrentDateTime; 	END_IF

IF bAutoStartPb AND ARbStnBasketAvailibilityRE[5].Q 	THEN ARbStnBasketInActivate[5] 	:= TRUE; ARsStnBasketInTime[5] := DSLocalSystemTimeML.sCurrentDateTime;
ARiStnBasketProductRecipeBuffer[5] 	:= DSStnBasketInfo[5].iProductRecipeNo; ARsStnBasketNoBuffer[5] 	:= DSStnBasketInfo[5].sReservedInt; 	END_IF

IF bAutoStartPb AND ARbStnBasketAvailibilityFE[5].Q 	THEN ARbStnBasketOutActivate[5] 	:= TRUE; ARsStnBasketOutTime[5] := DSLocalSystemTimeML.sCurrentDateTime; 	END_IF

IF bAutoStartPb AND ARbStnBasketAvailibilityRE[6].Q 	THEN ARbStnBasketInActivate[6] 	:= TRUE; ARsStnBasketInTime[6] := DSLocalSystemTimeML.sCurrentDateTime;
ARiStnBasketProductRecipeBuffer[6] 	:= DSStnBasketInfo[6].iProductRecipeNo; ARsStnBasketNoBuffer[6] 	:= DSStnBasketInfo[6].sReservedInt; 	END_IF

IF bAutoStartPb AND ARbStnBasketAvailibilityFE[6].Q 	THEN ARbStnBasketOutActivate[6] 	:= TRUE; ARsStnBasketOutTime[6] := DSLocalSystemTimeML.sCurrentDateTime; 	END_IF

IF bAutoStartPb AND ARbStnBasketAvailibilityRE[7].Q 	THEN ARbStnBasketInActivate[7] 	:= TRUE; ARsStnBasketInTime[7] := DSLocalSystemTimeML.sCurrentDateTime;
ARiStnBasketProductRecipeBuffer[7] 	:= DSStnBasketInfo[7].iProductRecipeNo; ARsStnBasketNoBuffer[7] 	:= DSStnBasketInfo[7].sReservedInt; 	END_IF

IF bAutoStartPb AND ARbStnBasketAvailibilityFE[7].Q 	THEN ARbStnBasketOutActivate[7] 	:= TRUE; ARsStnBasketOutTime[7] := DSLocalSystemTimeML.sCurrentDateTime; 	END_IF

